LIN {X 0,Y 445.396,Z 554.606,A -85,B 0,C 180,E1 -8729.095,E2 -8729.095} C_VEL
LIN {X 0,Y 445.404,Z 554.809,A -85,B 0,C 180,E1 -8729.999,E2 -8729.999} C_VEL
LIN {X 0,Y 445.396,Z 554.569,A -85,B 0,C 180,E1 -8730.903,E2 -8730.903} C_VEL
LIN {X 0,Y 445.399,Z 553.92,A -85,B 0,C 180,E1 -8731.808,E2 -8731.808} C_VEL
LIN {X 0,Y 445.449,Z 552.858,A -85,B 0,C 180,E1 -8732.712,E2 -8732.712} C_VEL
LIN {X 0,Y 445.409,Z 551.31,A -85,B 0,C 180,E1 -8733.618,E2 -8733.618} C_VEL
LIN {X 0,Y 445.481,Z 548.159,A -85,B 0,C 180,E1 -8734.977,E2 -8734.977} C_VEL
LIN {X 0,Y 445.529,Z 543.719,A -85,B 0,C 180,E1 -8736.385,E2 -8736.385} C_VEL
LIN {X 0,Y 445.7,Z 537.341,A -85,B 0,C 180,E1 -8737.93,E2 -8737.93} C_VEL
LIN {X 0,Y 445.942,Z 530.169,A -85,B 0,C 180,E1 -8739.295,E2 -8739.295} C_VEL
LIN {X 0,Y 446.309,Z 521.18,A -85,B 0,C 180,E1 -8740.662,E2 -8740.662} C_VEL
LIN {X 0,Y 446.885,Z 510.146,A -85,B 0,C 180,E1 -8742.026,E2 -8742.026} C_VEL
LIN {X 0,Y 447.422,Z 499.999,A -85,B 0,C 180,E1 -8743.042,E2 -8743.042} C_VEL
LIN {X 0,Y 447.933,Z 488.57,A -85,B 0,C 180,E1 -8743.958,E2 -8743.958} C_VEL
LIN {X 0,Y 448.567,Z 476.728,A -85,B 0,C 180,E1 -8744.691,E2 -8744.691} C_VEL
LIN {X 0,Y 448.997,Z 463.55,A -85,B 0,C 180,E1 -8745.286,E2 -8745.286} C_VEL
LIN {X 0,Y 449.466,Z 450.413,A -85,B 0,C 180,E1 -8745.676,E2 -8745.676} C_VEL
LIN {X 0,Y 450.087,Z 387.141,A -85,B 0,C 180,E1 -8746.743,E2 -8746.743} C_VEL
LIN {X 0,Y 450.275,Z 363.231,A -85,B 0,C 180,E1 -8747.197,E2 -8747.197} C_VEL
LIN {X 0,Y 447.374,Z 342.684,A -85,B 0,C 180,E1 -8747.702,E2 -8747.702} C_VEL
LIN {X 0,Y 448.31,Z 323.245,A -85,B 0,C 180,E1 -8751.134,E2 -8751.134} C_VEL
LIN {X 0,Y 449.367,Z 304.806,A -85,B 0,C 180,E1 -8754.441,E2 -8754.441} C_VEL
LIN {X 0,Y 447.45,Z 294.39,A -85,B 0,C 180,E1 -8756.454,E2 -8756.454} C_VEL
LIN {X 0,Y 446.525,Z 289.866,A -85,B 0,C 180,E1 -8757.378,E2 -8757.378} C_VEL
LIN {X 0,Y 446.425,Z 289.878,A -85,B 0,C 180,E1 -8760.249,E2 -8760.249} C_VEL
LIN {X 0,Y 446.442,Z 289.872,A -85,B 0,C 180,E1 -8763.453,E2 -8763.453} C_VEL
LIN {X 0,Y 446.396,Z 289.877,A -85,B 0,C 180,E1 -8766.744,E2 -8766.744} C_VEL
LIN {X 0,Y 446.431,Z 289.875,A -85,B 0,C 180,E1 -8770.198,E2 -8770.198} C_VEL
LIN {X 0,Y 446.393,Z 289.881,A -85,B 0,C 180,E1 -8773.596,E2 -8773.596} C_VEL
LIN {X 0,Y 446.391,Z 289.878,A -85,B 0,C 180,E1 -8776.403,E2 -8776.403} C_VEL
LIN {X 0,Y 446.398,Z 289.878,A -85,B 0,C 180,E1 -8779.085,E2 -8779.085} C_VEL
LIN {X 0,Y 446.399,Z 289.878,A -85,B 0,C 180,E1 -8782.12,E2 -8782.12} C_VEL
LIN {X 0,Y 446.416,Z 289.88,A -85,B 0,C 180,E1 -8785.476,E2 -8785.476} C_VEL
LIN {X 0,Y 446.406,Z 289.876,A -85,B 0,C 180,E1 -8788.699,E2 -8788.699} C_VEL
LIN {X 0,Y 446.415,Z 289.877,A -85,B 0,C 180,E1 -8791.836,E2 -8791.836} C_VEL
LIN {X 0,Y 446.422,Z 289.876,A -85,B 0,C 180,E1 -8794.845,E2 -8794.845} C_VEL
LIN {X 0,Y 446.439,Z 289.873,A -85,B 0,C 180,E1 -8798.245,E2 -8798.245} C_VEL
LIN {X 0,Y 446.441,Z 289.874,A -85,B 0,C 180,E1 -8801.648,E2 -8801.648} C_VEL
LIN {X 0,Y 446.495,Z 289.866,A -85,B 0,C 180,E1 -8804.479,E2 -8804.479} C_VEL
LIN {X 0,Y 446.506,Z 289.865,A -85,B 0,C 180,E1 -8808.193,E2 -8808.193} C_VEL
LIN {X 0,Y 446.519,Z 289.867,A -85,B 0,C 180,E1 -8810.944,E2 -8810.944} C_VEL
LIN {X 0,Y 446.588,Z 289.855,A -85,B 0,C 180,E1 -8813.675,E2 -8813.675} C_VEL
LIN {X 0,Y 446.651,Z 289.848,A -85,B 0,C 180,E1 -8817.294,E2 -8817.294} C_VEL
LIN {X 0,Y 446.686,Z 289.843,A -85,B 0,C 180,E1 -8820,E2 -8820} C_VEL
LIN {X 0,Y 446.64,Z 289.851,A -85,B 0,C 180,E1 -8822.706,E2 -8822.706} C_VEL
LIN {X 0,Y 446.595,Z 289.855,A -85,B 0,C 180,E1 -8826.324,E2 -8826.324} C_VEL
LIN {X 0,Y 446.515,Z 289.865,A -85,B 0,C 180,E1 -8829.056,E2 -8829.056} C_VEL
LIN {X 0,Y 446.513,Z 289.867,A -85,B 0,C 180,E1 -8832.73,E2 -8832.73} C_VEL
LIN {X 0,Y 446.479,Z 289.871,A -85,B 0,C 180,E1 -8836.46,E2 -8836.46} C_VEL
LIN {X 0,Y 446.459,Z 289.873,A -85,B 0,C 180,E1 -8839.304,E2 -8839.304} C_VEL
LIN {X 0,Y 446.41,Z 289.879,A -85,B 0,C 180,E1 -8842.2,E2 -8842.2} C_VEL
LIN {X 0,Y 446.431,Z 289.877,A -85,B 0,C 180,E1 -8845.154,E2 -8845.154} C_VEL
LIN {X 0,Y 446.432,Z 289.877,A -85,B 0,C 180,E1 -8848.182,E2 -8848.182} C_VEL
LIN {X 0,Y 446.408,Z 289.879,A -85,B 0,C 180,E1 -8851.301,E2 -8851.301} C_VEL
LIN {X 0,Y 446.422,Z 289.877,A -85,B 0,C 180,E1 -8854.524,E2 -8854.524} C_VEL
LIN {X 0,Y 446.405,Z 289.88,A -85,B 0,C 180,E1 -8858.079,E2 -8858.079} C_VEL
LIN {X 0,Y 446.416,Z 289.879,A -85,B 0,C 180,E1 -8860.918,E2 -8860.918} C_VEL
LIN {X 0,Y 446.393,Z 289.881,A -85,B 0,C 180,E1 -8863.847,E2 -8863.847} C_VEL
LIN {X 0,Y 446.392,Z 289.881,A -85,B 0,C 180,E1 -8866.405,E2 -8866.405} C_VEL
LIN {X 0,Y 446.423,Z 289.876,A -85,B 0,C 180,E1 -8869.083,E2 -8869.083} C_VEL
LIN {X 0,Y 446.405,Z 289.879,A -85,B 0,C 180,E1 -8872.122,E2 -8872.122} C_VEL
LIN {X 0,Y 446.42,Z 289.876,A -85,B 0,C 180,E1 -8875.478,E2 -8875.478} C_VEL
LIN {X 0,Y 446.413,Z 289.879,A -85,B 0,C 180,E1 -8878.701,E2 -8878.701} C_VEL
LIN {X 0,Y 446.483,Z 289.869,A -85,B 0,C 180,E1 -8881.822,E2 -8881.822} C_VEL
LIN {X 0,Y 446.448,Z 289.873,A -85,B 0,C 180,E1 -8884.848,E2 -8884.848} C_VEL
LIN {X 0,Y 446.448,Z 289.875,A -85,B 0,C 180,E1 -8888.246,E2 -8888.246} C_VEL
LIN {X 0,Y 446.519,Z 289.866,A -85,B 0,C 180,E1 -8891.653,E2 -8891.653} C_VEL
LIN {X 0,Y 447.511,Z 295.536,A -85,B 0,C 180,E1 -8892.133,E2 -8892.133} C_VEL
LIN {X 0,Y 451.074,Z 318.693,A -85,B 0,C 180,E1 -8892.665,E2 -8892.665} C_VEL
LIN {X 0,Y 450.362,Z 395.766,A -85,B 0,C 180,E1 -8893.901,E2 -8893.901} C_VEL
LIN {X 0,Y 449.639,Z 401.622,A -85,B 0,C 180,E1 -8893.969,E2 -8893.969} C_VEL
LIN {X 0,Y 445.281,Z 414.821,A -85,B 0,C 180,E1 -8894.091,E2 -8894.091} C_VEL
LIN {X 0,Y 443.656,Z 420.458,A -85,B 0,C 180,E1 -8894.209,E2 -8894.209} C_VEL
LIN {X 0,Y 442.987,Z 426.107,A -85,B 0,C 180,E1 -8894.404,E2 -8894.404} C_VEL
LIN {X 0,Y 442.505,Z 438.201,A -85,B 0,C 180,E1 -8894.986,E2 -8894.986} C_VEL
LIN {X 0,Y 442.002,Z 449.785,A -85,B 0,C 180,E1 -8895.734,E2 -8895.734} C_VEL
LIN {X 0,Y 441.476,Z 461.067,A -85,B 0,C 180,E1 -8896.674,E2 -8896.674} C_VEL
LIN {X 0,Y 440.791,Z 471.918,A -85,B 0,C 180,E1 -8897.805,E2 -8897.805} C_VEL
LIN {X 0,Y 440.215,Z 480.764,A -85,B 0,C 180,E1 -8898.956,E2 -8898.956} C_VEL
LIN {X 0,Y 439.7,Z 489.38,A -85,B 0,C 180,E1 -8900.339,E2 -8900.339} C_VEL
LIN {X 0,Y 439.185,Z 496.313,A -85,B 0,C 180,E1 -8901.72,E2 -8901.72} C_VEL
LIN {X 0,Y 438.904,Z 501.856,A -85,B 0,C 180,E1 -8903.114,E2 -8903.114} C_VEL
LIN {X 0,Y 438.627,Z 506.14,A -85,B 0,C 180,E1 -8904.484,E2 -8904.484} C_VEL
LIN {X 0,Y 438.529,Z 508.41,A -85,B 0,C 180,E1 -8905.405,E2 -8905.405} C_VEL
LIN {X 0,Y 438.578,Z 510.257,A -85,B 0,C 180,E1 -8906.326,E2 -8906.326} C_VEL
LIN {X 0,Y 438.457,Z 511.678,A -85,B 0,C 180,E1 -8907.245,E2 -8907.245} C_VEL
LIN {X 0,Y 438.312,Z 513.288,A -85,B 0,C 180,E1 -8909.082,E2 -8909.082} C_VEL
LIN {X 0,Y 438.314,Z 513.523,A -85,B 0,C 180,E1 -8910.001,E2 -8910.001} C_VEL
LIN {X 0,Y 438.354,Z 512.752,A -85,B 0,C 180,E1 -8911.838,E2 -8911.838} C_VEL
LIN {X 0,Y 438.457,Z 511.788,A -85,B 0,C 180,E1 -8912.757,E2 -8912.757} C_VEL
LIN {X 0,Y 438.572,Z 510.429,A -85,B 0,C 180,E1 -8913.676,E2 -8913.676} C_VEL
LIN {X 0,Y 438.531,Z 507.58,A -85,B 0,C 180,E1 -8915.058,E2 -8915.058} C_VEL
LIN {X 0,Y 438.877,Z 503.69,A -85,B 0,C 180,E1 -8916.437,E2 -8916.437} C_VEL
LIN {X 0,Y 439.039,Z 498.669,A -85,B 0,C 180,E1 -8917.821,E2 -8917.821} C_VEL
LIN {X 0,Y 439.469,Z 492.327,A -85,B 0,C 180,E1 -8919.203,E2 -8919.203} C_VEL
LIN {X 0,Y 439.967,Z 484.438,A -85,B 0,C 180,E1 -8920.586,E2 -8920.586} C_VEL
LIN {X 0,Y 440.452,Z 476.372,A -85,B 0,C 180,E1 -8921.739,E2 -8921.739} C_VEL
LIN {X 0,Y 441.183,Z 466.467,A -85,B 0,C 180,E1 -8922.887,E2 -8922.887} C_VEL
LIN {X 0,Y 441.757,Z 454.932,A -85,B 0,C 180,E1 -8923.96,E2 -8923.96} C_VEL
LIN {X 0,Y 442.266,Z 444.447,A -85,B 0,C 180,E1 -8924.73,E2 -8924.73} C_VEL
LIN {X 0,Y 442.742,Z 432.204,A -85,B 0,C 180,E1 -8925.42,E2 -8925.42} C_VEL
LIN {X 0,Y 443.237,Z 418.659,A -85,B 0,C 180,E1 -8925.963,E2 -8925.963} C_VEL
LIN {X 0,Y 443.407,Z 406.073,A -85,B 0,C 180,E1 -8926.282,E2 -8926.282} C_VEL
LIN {X 0,Y 444.227,Z 319.296,A -85,B 0,C 180,E1 -8927.699,E2 -8927.699} C_VEL
LIN {X 0,Y 440.588,Z 295.599,A -85,B 0,C 180,E1 -8928.263,E2 -8928.263} C_VEL
LIN {X 0,Y 439.49,Z 290.742,A -85,B 0,C 180,E1 -8928.699,E2 -8928.699} C_VEL
LIN {X 0,Y 439.394,Z 290.754,A -85,B 0,C 180,E1 -8931.921,E2 -8931.921} C_VEL
LIN {X 0,Y 439.415,Z 290.749,A -85,B 0,C 180,E1 -8934.573,E2 -8934.573} C_VEL
LIN {X 0,Y 439.445,Z 290.749,A -85,B 0,C 180,E1 -8937.633,E2 -8937.633} C_VEL
LIN {X 0,Y 439.366,Z 290.754,A -85,B 0,C 180,E1 -8940.789,E2 -8940.789} C_VEL
LIN {X 0,Y 439.389,Z 290.752,A -85,B 0,C 180,E1 -8944.044,E2 -8944.044} C_VEL
LIN {X 0,Y 439.353,Z 290.756,A -85,B 0,C 180,E1 -8946.887,E2 -8946.887} C_VEL
LIN {X 0,Y 439.411,Z 290.749,A -85,B 0,C 180,E1 -8949.85,E2 -8949.85} C_VEL
LIN {X 0,Y 439.39,Z 290.751,A -85,B 0,C 180,E1 -8952.628,E2 -8952.628} C_VEL
LIN {X 0,Y 439.407,Z 290.753,A -85,B 0,C 180,E1 -8955.271,E2 -8955.271} C_VEL
LIN {X 0,Y 439.394,Z 290.751,A -85,B 0,C 180,E1 -8958.744,E2 -8958.744} C_VEL
LIN {X 0,Y 439.379,Z 290.752,A -85,B 0,C 180,E1 -8961.608,E2 -8961.608} C_VEL
LIN {X 0,Y 439.404,Z 290.753,A -85,B 0,C 180,E1 -8964.844,E2 -8964.844} C_VEL
LIN {X 0,Y 439.378,Z 290.751,A -85,B 0,C 180,E1 -8968.14,E2 -8968.14} C_VEL
LIN {X 0,Y 439.437,Z 290.744,A -85,B 0,C 180,E1 -8971.598,E2 -8971.598} C_VEL
LIN {X 0,Y 439.393,Z 290.752,A -85,B 0,C 180,E1 -8974.414,E2 -8974.414} C_VEL
LIN {X 0,Y 439.369,Z 290.752,A -85,B 0,C 180,E1 -8977.425,E2 -8977.425} C_VEL
LIN {X 0,Y 439.458,Z 290.872,A -85,B 0,C 180,E1 -8979.247,E2 -8979.247} C_VEL
LIN {X 0,Y 440.572,Z 297.687,A -85,B 0,C 180,E1 -8980.912,E2 -8980.912} C_VEL
LIN {X 0,Y 440.519,Z 303.107,A -85,B 0,C 180,E1 -8982.174,E2 -8982.174} C_VEL
LIN {X 0,Y 443.779,Z 320.199,A -85,B 0,C 180,E1 -8982.629,E2 -8982.629} C_VEL
LIN {X 0,Y 442.424,Z 410.602,A -85,B 0,C 180,E1 -8984.362,E2 -8984.362} C_VEL
LIN {X 0,Y 442.117,Z 424.604,A -85,B 0,C 180,E1 -8984.824,E2 -8984.824} C_VEL
LIN {X 0,Y 441.633,Z 437.177,A -85,B 0,C 180,E1 -8985.426,E2 -8985.426} C_VEL
LIN {X 0,Y 441.219,Z 448.876,A -85,B 0,C 180,E1 -8986.177,E2 -8986.177} C_VEL
LIN {X 0,Y 440.784,Z 460.248,A -85,B 0,C 180,E1 -8987.102,E2 -8987.102} C_VEL
LIN {X 0,Y 440.285,Z 470.498,A -85,B 0,C 180,E1 -8988.14,E2 -8988.14} C_VEL
LIN {X 0,Y 439.756,Z 480.584,A -85,B 0,C 180,E1 -8989.409,E2 -8989.409} C_VEL
LIN {X 0,Y 439.38,Z 488.085,A -85,B 0,C 180,E1 -8990.564,E2 -8990.564} C_VEL
LIN {X 0,Y 438.995,Z 495.45,A -85,B 0,C 180,E1 -8991.947,E2 -8991.947} C_VEL
LIN {X 0,Y 438.781,Z 501.004,A -85,B 0,C 180,E1 -8993.251,E2 -8993.251} C_VEL
LIN {X 0,Y 438.617,Z 505.222,A -85,B 0,C 180,E1 -8994.483,E2 -8994.483} C_VEL
LIN {X 0,Y 438.545,Z 508.87,A -85,B 0,C 180,E1 -8995.864,E2 -8995.864} C_VEL
LIN {X 0,Y 438.457,Z 511.47,A -85,B 0,C 180,E1 -8997.244,E2 -8997.244} C_VEL
LIN {X 0,Y 438.354,Z 512.65,A -85,B 0,C 180,E1 -8998.162,E2 -8998.162} C_VEL
LIN {X 0,Y 438.313,Z 513.401,A -85,B 0,C 180,E1 -8999.081,E2 -8999.081} C_VEL
LIN {X 0,Y 438.317,Z 513.75,A -85,B 0,C 180,E1 -9000,E2 -9000} C_VEL
LIN {X 0,Y 438.342,Z 513.684,A -85,B 0,C 180,E1 -9000.919,E2 -9000.919} C_VEL
LIN {X 0,Y 438.391,Z 513.16,A -85,B 0,C 180,E1 -9001.837,E2 -9001.837} C_VEL
LIN {X 0,Y 438.468,Z 512.228,A -85,B 0,C 180,E1 -9002.756,E2 -9002.756} C_VEL
LIN {X 0,Y 438.588,Z 510.886,A -85,B 0,C 180,E1 -9003.675,E2 -9003.675} C_VEL
LIN {X 0,Y 438.566,Z 508.017,A -85,B 0,C 180,E1 -9005.056,E2 -9005.056} C_VEL
LIN {X 0,Y 438.911,Z 504.057,A -85,B 0,C 180,E1 -9006.436,E2 -9006.436} C_VEL
LIN {X 0,Y 439.14,Z 497.926,A -85,B 0,C 180,E1 -9008.05,E2 -9008.05} C_VEL
LIN {X 0,Y 439.579,Z 491.187,A -85,B 0,C 180,E1 -9009.432,E2 -9009.432} C_VEL
LIN {X 0,Y 440.085,Z 482.787,A -85,B 0,C 180,E1 -9010.815,E2 -9010.815} C_VEL
LIN {X 0,Y 440.469,Z 474.111,A -85,B 0,C 180,E1 -9011.971,E2 -9011.971} C_VEL
LIN {X 0,Y 441.135,Z 463.913,A -85,B 0,C 180,E1 -9013.074,E2 -9013.074} C_VEL
LIN {X 0,Y 441.704,Z 453.145,A -85,B 0,C 180,E1 -9014.019,E2 -9014.019} C_VEL
LIN {X 0,Y 442.222,Z 441.072,A -85,B 0,C 180,E1 -9014.849,E2 -9014.849} C_VEL
LIN {X 0,Y 442.776,Z 427.768,A -85,B 0,C 180,E1 -9015.536,E2 -9015.536} C_VEL
LIN {X 0,Y 443.111,Z 415.088,A -85,B 0,C 180,E1 -9015.996,E2 -9015.996} C_VEL
LIN {X 0,Y 443.534,Z 392.837,A -85,B 0,C 180,E1 -9016.483,E2 -9016.483} C_VEL
LIN {X 0,Y 445.167,Z 320.736,A -85,B 0,C 180,E1 -9017.995,E2 -9017.995} C_VEL
LIN {X 0,Y 441.629,Z 306.236,A -85,B 0,C 180,E1 -9018.559,E2 -9018.559} C_VEL
LIN {X 0,Y 441.447,Z 300.594,A -85,B 0,C 180,E1 -9020.064,E2 -9020.064} C_VEL
LIN {X 0,Y 439.704,Z 292.144,A -85,B 0,C 180,E1 -9022.557,E2 -9022.557} C_VEL
LIN {X 0,Y 439.393,Z 290.755,A -85,B 0,C 180,E1 -9023.009,E2 -9023.009} C_VEL
LIN {X 0,Y 439.37,Z 290.758,A -85,B 0,C 180,E1 -9026.393,E2 -9026.393} C_VEL
LIN {X 0,Y 439.38,Z 290.756,A -85,B 0,C 180,E1 -9028.676,E2 -9028.676} C_VEL
LIN {X 0,Y 439.345,Z 290.758,A -85,B 0,C 180,E1 -9032.024,E2 -9032.024} C_VEL
LIN {X 0,Y 439.385,Z 290.754,A -85,B 0,C 180,E1 -9035.337,E2 -9035.337} C_VEL
LIN {X 0,Y 439.356,Z 290.758,A -85,B 0,C 180,E1 -9038.598,E2 -9038.598} C_VEL
LIN {X 0,Y 439.366,Z 290.755,A -85,B 0,C 180,E1 -9041.252,E2 -9041.252} C_VEL
LIN {X 0,Y 439.377,Z 290.757,A -85,B 0,C 180,E1 -9044.733,E2 -9044.733} C_VEL
LIN {X 0,Y 439.35,Z 290.757,A -85,B 0,C 180,E1 -9047.789,E2 -9047.789} C_VEL
LIN {X 0,Y 439.361,Z 290.755,A -85,B 0,C 180,E1 -9051.402,E2 -9051.402} C_VEL
LIN {X 0,Y 439.401,Z 290.753,A -85,B 0,C 180,E1 -9054.843,E2 -9054.843} C_VEL
LIN {X 0,Y 439.376,Z 290.761,A -85,B 0,C 180,E1 -9058.139,E2 -9058.139} C_VEL
LIN {X 0,Y 439.437,Z 290.78,A -85,B 0,C 180,E1 -9061.327,E2 -9061.327} C_VEL
LIN {X 0,Y 441.863,Z 301.055,A -85,B 0,C 180,E1 -9063.808,E2 -9063.808} C_VEL
LIN {X 0,Y 442.928,Z 307.495,A -85,B 0,C 180,E1 -9065.234,E2 -9065.234} C_VEL
LIN {X 0,Y 441.744,Z 323.154,A -85,B 0,C 180,E1 -9068.29,E2 -9068.29} C_VEL
LIN {X 0,Y 440.732,Z 339.974,A -85,B 0,C 180,E1 -9071.42,E2 -9071.42} C_VEL
LIN {X 0,Y 443.63,Z 357.852,A -85,B 0,C 180,E1 -9071.993,E2 -9071.993} C_VEL
LIN {X 0,Y 444.532,Z 366.532,A -85,B 0,C 180,E1 -9072.239,E2 -9072.239} C_VEL
LIN {X 0,Y 442.866,Z 451.22,A -85,B 0,C 180,E1 -9073.994,E2 -9073.994} C_VEL
LIN {X 0,Y 442.319,Z 464.599,A -85,B 0,C 180,E1 -9074.446,E2 -9074.446} C_VEL
LIN {X 0,Y 441.749,Z 476.41,A -85,B 0,C 180,E1 -9075.016,E2 -9075.016} C_VEL
LIN {X 0,Y 441.114,Z 488.934,A -85,B 0,C 180,E1 -9075.82,E2 -9075.82} C_VEL
LIN {X 0,Y 440.507,Z 499.92,A -85,B 0,C 180,E1 -9076.709,E2 -9076.709} C_VEL
LIN {X 0,Y 439.924,Z 510.52,A -85,B 0,C 180,E1 -9077.779,E2 -9077.779} C_VEL
LIN {X 0,Y 439.448,Z 519.842,A -85,B 0,C 180,E1 -9078.935,E2 -9078.935} C_VEL
LIN {X 0,Y 438.971,Z 528.974,A -85,B 0,C 180,E1 -9080.321,E2 -9080.321} C_VEL
LIN {X 0,Y 438.667,Z 536.272,A -85,B 0,C 180,E1 -9081.709,E2 -9081.709} C_VEL
LIN {X 0,Y 438.46,Z 542.113,A -85,B 0,C 180,E1 -9083.095,E2 -9083.095} C_VEL
LIN {X 0,Y 438.392,Z 546.704,A -85,B 0,C 180,E1 -9084.479,E2 -9084.479} C_VEL
LIN {X 0,Y 438.35,Z 549.141,A -85,B 0,C 180,E1 -9085.401,E2 -9085.401} C_VEL
LIN {X 0,Y 438.294,Z 551.105,A -85,B 0,C 180,E1 -9086.322,E2 -9086.322} C_VEL
LIN {X 0,Y 438.373,Z 552.583,A -85,B 0,C 180,E1 -9087.242,E2 -9087.242} C_VEL
LIN {X 0,Y 438.319,Z 553.638,A -85,B 0,C 180,E1 -9088.161,E2 -9088.161} C_VEL
LIN {X 0,Y 438.306,Z 554.281,A -85,B 0,C 180,E1 -9089.08,E2 -9089.08} C_VEL
LIN {X 0,Y 438.325,Z 554.464,A -85,B 0,C 180,E1 -9089.999,E2 -9089.999} C_VEL
LIN {X 0,Y 438.306,Z 554.212,A -85,B 0,C 180,E1 -9090.918,E2 -9090.918} C_VEL
LIN {X 0,Y 438.319,Z 553.55,A -85,B 0,C 180,E1 -9091.837,E2 -9091.837} C_VEL
LIN {X 0,Y 438.375,Z 552.466,A -85,B 0,C 180,E1 -9092.756,E2 -9092.756} C_VEL
LIN {X 0,Y 438.312,Z 549.968,A -85,B 0,C 180,E1 -9094.137,E2 -9094.137} C_VEL
LIN {X 0,Y 438.383,Z 546.416,A -85,B 0,C 180,E1 -9095.519,E2 -9095.519} C_VEL
LIN {X 0,Y 438.494,Z 541.701,A -85,B 0,C 180,E1 -9096.903,E2 -9096.903} C_VEL
LIN {X 0,Y 438.668,Z 535.673,A -85,B 0,C 180,E1 -9098.289,E2 -9098.289} C_VEL
LIN {X 0,Y 438.94,Z 528.137,A -85,B 0,C 180,E1 -9099.677,E2 -9099.677} C_VEL
LIN {X 0,Y 439.474,Z 517.318,A -85,B 0,C 180,E1 -9101.296,E2 -9101.296} C_VEL
LIN {X 0,Y 439.999,Z 507.714,A -85,B 0,C 180,E1 -9102.452,E2 -9102.452} C_VEL
LIN {X 0,Y 440.662,Z 496.446,A -85,B 0,C 180,E1 -9103.541,E2 -9103.541} C_VEL
LIN {X 0,Y 441.217,Z 484.939,A -85,B 0,C 180,E1 -9104.411,E2 -9104.411} C_VEL
LIN {X 0,Y 441.88,Z 471.957,A -85,B 0,C 180,E1 -9105.154,E2 -9105.154} C_VEL
LIN {X 0,Y 442.338,Z 460.172,A -85,B 0,C 180,E1 -9105.64,E2 -9105.64} C_VEL
LIN {X 0,Y 442.695,Z 447.345,A -85,B 0,C 180,E1 -9105.981,E2 -9105.981} C_VEL
LIN {X 0,Y 443.419,Z 376.801,A -85,B 0,C 180,E1 -9107.158,E2 -9107.158} C_VEL
LIN {X 0,Y 443.415,Z 363.933,A -85,B 0,C 180,E1 -9107.412,E2 -9107.412} C_VEL
LIN {X 0,Y 440.389,Z 342.46,A -85,B 0,C 180,E1 -9107.947,E2 -9107.947} C_VEL
LIN {X 0,Y 441.313,Z 324.12,A -85,B 0,C 180,E1 -9111.24,E2 -9111.24} C_VEL
LIN {X 0,Y 442.378,Z 306.746,A -85,B 0,C 180,E1 -9114.396,E2 -9114.396} C_VEL
LIN {X 0,Y 441.381,Z 299.941,A -85,B 0,C 180,E1 -9115.714,E2 -9115.714} C_VEL
LIN {X 0,Y 439.484,Z 290.743,A -85,B 0,C 180,E1 -9117.564,E2 -9117.564} C_VEL
LIN {X 0,Y 439.358,Z 290.753,A -85,B 0,C 180,E1 -9120.787,E2 -9120.787} C_VEL
LIN {X 0,Y 439.384,Z 290.756,A -85,B 0,C 180,E1 -9124.043,E2 -9124.043} C_VEL
LIN {X 0,Y 439.342,Z 290.755,A -85,B 0,C 180,E1 -9126.886,E2 -9126.886} C_VEL
LIN {X 0,Y 439.397,Z 290.755,A -85,B 0,C 180,E1 -9129.848,E2 -9129.848} C_VEL
LIN {X 0,Y 439.365,Z 290.753,A -85,B 0,C 180,E1 -9132.624,E2 -9132.624} C_VEL
LIN {X 0,Y 439.393,Z 290.751,A -85,B 0,C 180,E1 -9135.269,E2 -9135.269} C_VEL
LIN {X 0,Y 439.364,Z 290.753,A -85,B 0,C 180,E1 -9138.745,E2 -9138.745} C_VEL
LIN {X 0,Y 439.358,Z 290.76,A -85,B 0,C 180,E1 -9141.609,E2 -9141.609} C_VEL
LIN {X 0,Y 439.389,Z 290.75,A -85,B 0,C 180,E1 -9144.843,E2 -9144.843} C_VEL
LIN {X 0,Y 439.364,Z 290.755,A -85,B 0,C 180,E1 -9148.139,E2 -9148.139} C_VEL
LIN {X 0,Y 439.391,Z 290.754,A -85,B 0,C 180,E1 -9151.606,E2 -9151.606} C_VEL
LIN {X 0,Y 439.362,Z 290.754,A -85,B 0,C 180,E1 -9154.412,E2 -9154.412} C_VEL
LIN {X 0,Y 439.353,Z 290.759,A -85,B 0,C 180,E1 -9157.424,E2 -9157.424} C_VEL
LIN {X 0,Y 439.432,Z 290.746,A -85,B 0,C 180,E1 -9160.663,E2 -9160.663} C_VEL
LIN {X 0,Y 439.451,Z 290.744,A -85,B 0,C 180,E1 -9164.224,E2 -9164.224} C_VEL
LIN {X 0,Y 439.473,Z 290.742,A -85,B 0,C 180,E1 -9168.001,E2 -9168.001} C_VEL
LIN {X 0,Y 439.493,Z 290.739,A -85,B 0,C 180,E1 -9171.725,E2 -9171.725} C_VEL
LIN {X 0,Y 439.58,Z 290.728,A -85,B 0,C 180,E1 -9174.495,E2 -9174.495} C_VEL
LIN {X 0,Y 439.619,Z 290.723,A -85,B 0,C 180,E1 -9178.168,E2 -9178.168} C_VEL
LIN {X 0,Y 439.575,Z 290.732,A -85,B 0,C 180,E1 -9180.916,E2 -9180.916} C_VEL
LIN {X 0,Y 439.591,Z 290.73,A -85,B 0,C 180,E1 -9182.749,E2 -9182.749} C_VEL
LIN {X 0,Y 439.548,Z 290.733,A -85,B 0,C 180,E1 -9186.426,E2 -9186.426} C_VEL
LIN {X 0,Y 439.48,Z 290.742,A -85,B 0,C 180,E1 -9189.202,E2 -9189.202} C_VEL
LIN {X 0,Y 439.456,Z 290.745,A -85,B 0,C 180,E1 -9192.938,E2 -9192.938} C_VEL
LIN {X 0,Y 439.437,Z 290.747,A -85,B 0,C 180,E1 -9196.348,E2 -9196.348} C_VEL
LIN {X 0,Y 439.393,Z 290.752,A -85,B 0,C 180,E1 -9199.627,E2 -9199.627} C_VEL
LIN {X 0,Y 439.355,Z 290.758,A -85,B 0,C 180,E1 -9202.576,E2 -9202.576} C_VEL
LIN {X 0,Y 439.37,Z 290.754,A -85,B 0,C 180,E1 -9205.587,E2 -9205.587} C_VEL
LIN {X 0,Y 439.389,Z 290.753,A -85,B 0,C 180,E1 -9208.676,E2 -9208.676} C_VEL
LIN {X 0,Y 439.363,Z 290.756,A -85,B 0,C 180,E1 -9212.031,E2 -9212.031} C_VEL
LIN {X 0,Y 439.386,Z 290.753,A -85,B 0,C 180,E1 -9215.341,E2 -9215.341} C_VEL
LIN {X 0,Y 439.362,Z 290.757,A -85,B 0,C 180,E1 -9218.597,E2 -9218.597} C_VEL
LIN {X 0,Y 439.375,Z 290.754,A -85,B 0,C 180,E1 -9221.257,E2 -9221.257} C_VEL
LIN {X 0,Y 439.393,Z 290.754,A -85,B 0,C 180,E1 -9224.731,E2 -9224.731} C_VEL
LIN {X 0,Y 439.391,Z 290.753,A -85,B 0,C 180,E1 -9227.797,E2 -9227.797} C_VEL
LIN {X 0,Y 439.407,Z 290.751,A -85,B 0,C 180,E1 -9230.227,E2 -9230.227} C_VEL
LIN {X 0,Y 439.37,Z 290.755,A -85,B 0,C 180,E1 -9233.714,E2 -9233.714} C_VEL
LIN {X 0,Y 439.368,Z 290.754,A -85,B 0,C 180,E1 -9237.055,E2 -9237.055} C_VEL
LIN {X 0,Y 439.38,Z 290.755,A -85,B 0,C 180,E1 -9240.275,E2 -9240.275} C_VEL
LIN {X 0,Y 439.427,Z 290.747,A -85,B 0,C 180,E1 -9243.397,E2 -9243.397} C_VEL
LIN {X 0,Y 439.385,Z 290.756,A -85,B 0,C 180,E1 -9246.431,E2 -9246.431} C_VEL
LIN {X 0,Y 439.389,Z 290.753,A -85,B 0,C 180,E1 -9249.398,E2 -9249.398} C_VEL
LIN {X 0,Y 439.466,Z 290.745,A -85,B 0,C 180,E1 -9251.42,E2 -9251.42} C_VEL
LIN {X 0,Y 440.672,Z 296.048,A -85,B 0,C 180,E1 -9251.854,E2 -9251.854} C_VEL
LIN {X 0,Y 444.268,Z 319.368,A -85,B 0,C 180,E1 -9252.398,E2 -9252.398} C_VEL
LIN {X 0,Y 443.349,Z 409.998,A -85,B 0,C 180,E1 -9253.895,E2 -9253.895} C_VEL
LIN {X 0,Y 443.073,Z 423.507,A -85,B 0,C 180,E1 -9254.298,E2 -9254.298} C_VEL
LIN {X 0,Y 442.987,Z 426.107,A -85,B 0,C 180,E1 -9254.404,E2 -9254.404} C_VEL
LIN {X 0,Y 442.25,Z 431.718,A -85,B 0,C 180,E1 -9254.629,E2 -9254.629} C_VEL
LIN {X 0,Y 439.177,Z 440.702,A -85,B 0,C 180,E1 -9255.011,E2 -9255.011} C_VEL
LIN {X 0,Y 435.898,Z 449.345,A -85,B 0,C 180,E1 -9255.474,E2 -9255.474} C_VEL
LIN {X 0,Y 434.895,Z 454.419,A -85,B 0,C 180,E1 -9255.84,E2 -9255.84} C_VEL
LIN {X 0,Y 434.317,Z 465.893,A -85,B 0,C 180,E1 -9256.907,E2 -9256.907} C_VEL
LIN {X 0,Y 433.549,Z 476,A -85,B 0,C 180,E1 -9258.073,E2 -9258.073} C_VEL
LIN {X 0,Y 432.962,Z 485.619,A -85,B 0,C 180,E1 -9259.479,E2 -9259.479} C_VEL
LIN {X 0,Y 432.406,Z 493.357,A -85,B 0,C 180,E1 -9260.883,E2 -9260.883} C_VEL
LIN {X 0,Y 432.05,Z 498.592,A -85,B 0,C 180,E1 -9262.053,E2 -9262.053} C_VEL
LIN {X 0,Y 431.832,Z 503.702,A -85,B 0,C 180,E1 -9263.459,E2 -9263.459} C_VEL
LIN {X 0,Y 431.473,Z 507.664,A -85,B 0,C 180,E1 -9264.861,E2 -9264.861} C_VEL
LIN {X 0,Y 431.495,Z 510.575,A -85,B 0,C 180,E1 -9266.265,E2 -9266.265} C_VEL
LIN {X 0,Y 431.39,Z 511.994,A -85,B 0,C 180,E1 -9267.2,E2 -9267.2} C_VEL
LIN {X 0,Y 431.226,Z 513.604,A -85,B 0,C 180,E1 -9269.067,E2 -9269.067} C_VEL
LIN {X 0,Y 431.225,Z 513.839,A -85,B 0,C 180,E1 -9270.001,E2 -9270.001} C_VEL
LIN {X 0,Y 431.276,Z 513.068,A -85,B 0,C 180,E1 -9271.869,E2 -9271.869} C_VEL
LIN {X 0,Y 431.389,Z 512.103,A -85,B 0,C 180,E1 -9272.802,E2 -9272.802} C_VEL
LIN {X 0,Y 431.489,Z 510.744,A -85,B 0,C 180,E1 -9273.736,E2 -9273.736} C_VEL
LIN {X 0,Y 431.471,Z 507.895,A -85,B 0,C 180,E1 -9275.141,E2 -9275.141} C_VEL
LIN {X 0,Y 431.809,Z 504.005,A -85,B 0,C 180,E1 -9276.543,E2 -9276.543} C_VEL
LIN {X 0,Y 432.022,Z 498.981,A -85,B 0,C 180,E1 -9277.949,E2 -9277.949} C_VEL
LIN {X 0,Y 432.474,Z 492.638,A -85,B 0,C 180,E1 -9279.353,E2 -9279.353} C_VEL
LIN {X 0,Y 432.997,Z 484.746,A -85,B 0,C 180,E1 -9280.759,E2 -9280.759} C_VEL
LIN {X 0,Y 433.522,Z 476.678,A -85,B 0,C 180,E1 -9281.93,E2 -9281.93} C_VEL
LIN {X 0,Y 434.286,Z 466.768,A -85,B 0,C 180,E1 -9283.096,E2 -9283.096} C_VEL
LIN {X 0,Y 434.853,Z 455.78,A -85,B 0,C 180,E1 -9284.138,E2 -9284.138} C_VEL
LIN {X 0,Y 435.417,Z 444.736,A -85,B 0,C 180,E1 -9284.967,E2 -9284.967} C_VEL
LIN {X 0,Y 435.924,Z 432.478,A -85,B 0,C 180,E1 -9285.668,E2 -9285.668} C_VEL
LIN {X 0,Y 436.417,Z 419.742,A -85,B 0,C 180,E1 -9286.189,E2 -9286.189} C_VEL
LIN {X 0,Y 436.628,Z 407.793,A -85,B 0,C 180,E1 -9286.512,E2 -9286.512} C_VEL
LIN {X 0,Y 437.477,Z 319.891,A -85,B 0,C 180,E1 -9287.974,E2 -9287.974} C_VEL
LIN {X 0,Y 433.744,Z 296.583,A -85,B 0,C 180,E1 -9288.537,E2 -9288.537} C_VEL
LIN {X 0,Y 432.439,Z 291.679,A -85,B 0,C 180,E1 -9288.919,E2 -9288.919} C_VEL
LIN {X 0,Y 432.349,Z 291.63,A -85,B 0,C 180,E1 -9292.095,E2 -9292.095} C_VEL
LIN {X 0,Y 432.351,Z 291.628,A -85,B 0,C 180,E1 -9295.002,E2 -9295.002} C_VEL
LIN {X 0,Y 432.386,Z 291.625,A -85,B 0,C 180,E1 -9298.124,E2 -9298.124} C_VEL
LIN {X 0,Y 432.325,Z 291.634,A -85,B 0,C 180,E1 -9301.347,E2 -9301.347} C_VEL
LIN {X 0,Y 432.342,Z 291.628,A -85,B 0,C 180,E1 -9304.678,E2 -9304.678} C_VEL
LIN {X 0,Y 432.343,Z 291.629,A -85,B 0,C 180,E1 -9308.15,E2 -9308.15} C_VEL
LIN {X 0,Y 432.338,Z 291.631,A -85,B 0,C 180,E1 -9311.602,E2 -9311.602} C_VEL
LIN {X 0,Y 432.345,Z 291.627,A -85,B 0,C 180,E1 -9314.347,E2 -9314.347} C_VEL
LIN {X 0,Y 432.325,Z 291.634,A -85,B 0,C 180,E1 -9317.016,E2 -9317.016} C_VEL
LIN {X 0,Y 432.338,Z 291.629,A -85,B 0,C 180,E1 -9319.821,E2 -9319.821} C_VEL
LIN {X 0,Y 432.312,Z 291.638,A -85,B 0,C 180,E1 -9323.022,E2 -9323.022} C_VEL
LIN {X 0,Y 432.364,Z 291.625,A -85,B 0,C 180,E1 -9325.997,E2 -9325.997} C_VEL
LIN {X 0,Y 432.352,Z 291.627,A -85,B 0,C 180,E1 -9329.49,E2 -9329.49} C_VEL
LIN {X 0,Y 432.39,Z 291.626,A -85,B 0,C 180,E1 -9332.928,E2 -9332.928} C_VEL
LIN {X 0,Y 432.372,Z 291.624,A -85,B 0,C 180,E1 -9336.023,E2 -9336.023} C_VEL
LIN {X 0,Y 432.417,Z 291.788,A -85,B 0,C 180,E1 -9339.112,E2 -9339.112} C_VEL
LIN {X 0,Y 433.645,Z 299.803,A -85,B 0,C 180,E1 -9341.087,E2 -9341.087} C_VEL
LIN {X 0,Y 433.562,Z 303.369,A -85,B 0,C 180,E1 -9341.924,E2 -9341.924} C_VEL
LIN {X 0,Y 436.906,Z 321.998,A -85,B 0,C 180,E1 -9342.425,E2 -9342.425} C_VEL
LIN {X 0,Y 435.475,Z 411.691,A -85,B 0,C 180,E1 -9344.196,E2 -9344.196} C_VEL
LIN {X 0,Y 435.162,Z 425.405,A -85,B 0,C 180,E1 -9344.665,E2 -9344.665} C_VEL
LIN {X 0,Y 434.669,Z 437.301,A -85,B 0,C 180,E1 -9345.247,E2 -9345.247} C_VEL
LIN {X 0,Y 434.212,Z 450.31,A -85,B 0,C 180,E1 -9346.104,E2 -9346.104} C_VEL
LIN {X 0,Y 433.754,Z 461.089,A -85,B 0,C 180,E1 -9347.008,E2 -9347.008} C_VEL
LIN {X 0,Y 433.252,Z 471.224,A -85,B 0,C 180,E1 -9348.064,E2 -9348.064} C_VEL
LIN {X 0,Y 432.724,Z 480.421,A -85,B 0,C 180,E1 -9349.235,E2 -9349.235} C_VEL
LIN {X 0,Y 432.287,Z 489.401,A -85,B 0,C 180,E1 -9350.643,E2 -9350.643} C_VEL
LIN {X 0,Y 431.905,Z 496.537,A -85,B 0,C 180,E1 -9352.05,E2 -9352.05} C_VEL
LIN {X 0,Y 431.702,Z 502.243,A -85,B 0,C 180,E1 -9353.456,E2 -9353.456} C_VEL
LIN {X 0,Y 431.463,Z 506.706,A -85,B 0,C 180,E1 -9354.86,E2 -9354.86} C_VEL
LIN {X 0,Y 431.454,Z 510.047,A -85,B 0,C 180,E1 -9356.264,E2 -9356.264} C_VEL
LIN {X 0,Y 431.388,Z 511.719,A -85,B 0,C 180,E1 -9357.199,E2 -9357.199} C_VEL
LIN {X 0,Y 431.276,Z 512.942,A -85,B 0,C 180,E1 -9358.132,E2 -9358.132} C_VEL
LIN {X 0,Y 431.227,Z 513.715,A -85,B 0,C 180,E1 -9359.066,E2 -9359.066} C_VEL
LIN {X 0,Y 431.228,Z 514.086,A -85,B 0,C 180,E1 -9360,E2 -9360} C_VEL
LIN {X 0,Y 431.255,Z 514.048,A -85,B 0,C 180,E1 -9360.934,E2 -9360.934} C_VEL
LIN {X 0,Y 431.31,Z 513.549,A -85,B 0,C 180,E1 -9361.868,E2 -9361.868} C_VEL
LIN {X 0,Y 431.4,Z 512.631,A -85,B 0,C 180,E1 -9362.801,E2 -9362.801} C_VEL
LIN {X 0,Y 431.528,Z 511.305,A -85,B 0,C 180,E1 -9363.735,E2 -9363.735} C_VEL
LIN {X 0,Y 431.5,Z 508.469,A -85,B 0,C 180,E1 -9365.139,E2 -9365.139} C_VEL
LIN {X 0,Y 431.873,Z 504.539,A -85,B 0,C 180,E1 -9366.541,E2 -9366.541} C_VEL
LIN {X 0,Y 432.081,Z 499.45,A -85,B 0,C 180,E1 -9367.947,E2 -9367.947} C_VEL
LIN {X 0,Y 432.523,Z 492.98,A -85,B 0,C 180,E1 -9369.351,E2 -9369.351} C_VEL
LIN {X 0,Y 433.049,Z 484.897,A -85,B 0,C 180,E1 -9370.756,E2 -9370.756} C_VEL
LIN {X 0,Y 433.505,Z 476.637,A -85,B 0,C 180,E1 -9371.929,E2 -9371.929} C_VEL
LIN {X 0,Y 434.163,Z 466.5,A -85,B 0,C 180,E1 -9373.098,E2 -9373.098} C_VEL
LIN {X 0,Y 434.811,Z 455.525,A -85,B 0,C 180,E1 -9374.114,E2 -9374.114} C_VEL
LIN {X 0,Y 435.389,Z 443.971,A -85,B 0,C 180,E1 -9374.967,E2 -9374.967} C_VEL
LIN {X 0,Y 435.938,Z 431.516,A -85,B 0,C 180,E1 -9375.666,E2 -9375.666} C_VEL
LIN {X 0,Y 436.362,Z 418.694,A -85,B 0,C 180,E1 -9376.191,E2 -9376.191} C_VEL
LIN {X 0,Y 436.642,Z 405.669,A -85,B 0,C 180,E1 -9376.54,E2 -9376.54} C_VEL
LIN {X 0,Y 438.533,Z 326.572,A -85,B 0,C 180,E1 -9378.238,E2 -9378.238} C_VEL
LIN {X 0,Y 438.515,Z 321.194,A -85,B 0,C 180,E1 -9378.368,E2 -9378.368} C_VEL
LIN {X 0,Y 434.839,Z 306.813,A -85,B 0,C 180,E1 -9378.951,E2 -9378.951} C_VEL
LIN {X 0,Y 434.564,Z 302.02,A -85,B 0,C 180,E1 -9380.279,E2 -9380.279} C_VEL
LIN {X 0,Y 432.718,Z 293.276,A -85,B 0,C 180,E1 -9382.942,E2 -9382.942} C_VEL
LIN {X 0,Y 432.352,Z 291.633,A -85,B 0,C 180,E1 -9383.469,E2 -9383.469} C_VEL
LIN {X 0,Y 432.313,Z 291.637,A -85,B 0,C 180,E1 -9386.603,E2 -9386.603} C_VEL
LIN {X 0,Y 432.318,Z 291.636,A -85,B 0,C 180,E1 -9389.189,E2 -9389.189} C_VEL
LIN {X 0,Y 432.308,Z 291.636,A -85,B 0,C 180,E1 -9392.444,E2 -9392.444} C_VEL
LIN {X 0,Y 432.333,Z 291.631,A -85,B 0,C 180,E1 -9395.818,E2 -9395.818} C_VEL
LIN {X 0,Y 432.303,Z 291.635,A -85,B 0,C 180,E1 -9399.348,E2 -9399.348} C_VEL
LIN {X 0,Y 432.306,Z 291.634,A -85,B 0,C 180,E1 -9401.801,E2 -9401.801} C_VEL
LIN {X 0,Y 432.335,Z 291.632,A -85,B 0,C 180,E1 -9404.347,E2 -9404.347} C_VEL
LIN {X 0,Y 432.304,Z 291.635,A -85,B 0,C 180,E1 -9407.018,E2 -9407.018} C_VEL
LIN {X 0,Y 432.292,Z 291.637,A -85,B 0,C 180,E1 -9409.828,E2 -9409.828} C_VEL
LIN {X 0,Y 432.306,Z 291.636,A -85,B 0,C 180,E1 -9413.021,E2 -9413.021} C_VEL
LIN {X 0,Y 432.363,Z 291.631,A -85,B 0,C 180,E1 -9415.996,E2 -9415.996} C_VEL
LIN {X 0,Y 432.35,Z 291.637,A -85,B 0,C 180,E1 -9419.489,E2 -9419.489} C_VEL
LIN {X 0,Y 432.386,Z 291.75,A -85,B 0,C 180,E1 -9420.854,E2 -9420.854} C_VEL
LIN {X 0,Y 434.5,Z 300.489,A -85,B 0,C 180,E1 -9423.069,E2 -9423.069} C_VEL
LIN {X 0,Y 436.059,Z 308.799,A -85,B 0,C 180,E1 -9424.996,E2 -9424.996} C_VEL
LIN {X 0,Y 435.324,Z 318.485,A -85,B 0,C 180,E1 -9426.959,E2 -9426.959} C_VEL
LIN {X 0,Y 434.2,Z 333.348,A -85,B 0,C 180,E1 -9429.85,E2 -9429.85} C_VEL
LIN {X 0,Y 433.877,Z 339.369,A -85,B 0,C 180,E1 -9430.993,E2 -9430.993} C_VEL
LIN {X 0,Y 436.844,Z 356.926,A -85,B 0,C 180,E1 -9431.599,E2 -9431.599} C_VEL
LIN {X 0,Y 437.939,Z 367.347,A -85,B 0,C 180,E1 -9431.908,E2 -9431.908} C_VEL
LIN {X 0,Y 436.125,Z 450.293,A -85,B 0,C 180,E1 -9433.679,E2 -9433.679} C_VEL
LIN {X 0,Y 435.57,Z 463.723,A -85,B 0,C 180,E1 -9434.139,E2 -9434.139} C_VEL
LIN {X 0,Y 434.902,Z 476.616,A -85,B 0,C 180,E1 -9434.775,E2 -9434.775} C_VEL
LIN {X 0,Y 434.228,Z 489.007,A -85,B 0,C 180,E1 -9435.59,E2 -9435.59} C_VEL
LIN {X 0,Y 433.535,Z 500.715,A -85,B 0,C 180,E1 -9436.571,E2 -9436.571} C_VEL
LIN {X 0,Y 432.909,Z 511.4,A -85,B 0,C 180,E1 -9437.696,E2 -9437.696} C_VEL
LIN {X 0,Y 432.331,Z 521.361,A -85,B 0,C 180,E1 -9438.987,E2 -9438.987} C_VEL
LIN {X 0,Y 431.862,Z 530.071,A -85,B 0,C 180,E1 -9440.397,E2 -9440.397} C_VEL
LIN {X 0,Y 431.579,Z 537.099,A -85,B 0,C 180,E1 -9441.807,E2 -9441.807} C_VEL
LIN {X 0,Y 431.34,Z 543.533,A -85,B 0,C 180,E1 -9443.45,E2 -9443.45} C_VEL
LIN {X 0,Y 431.306,Z 547.722,A -85,B 0,C 180,E1 -9444.857,E2 -9444.857} C_VEL
LIN {X 0,Y 431.2,Z 550.81,A -85,B 0,C 180,E1 -9446.261,E2 -9446.261} C_VEL
LIN {X 0,Y 431.281,Z 552.28,A -85,B 0,C 180,E1 -9447.197,E2 -9447.197} C_VEL
LIN {X 0,Y 431.241,Z 553.326,A -85,B 0,C 180,E1 -9448.131,E2 -9448.131} C_VEL
LIN {X 0,Y 431.22,Z 553.955,A -85,B 0,C 180,E1 -9449.065,E2 -9449.065} C_VEL
LIN {X 0,Y 431.235,Z 554.115,A -85,B 0,C 180,E1 -9449.999,E2 -9449.999} C_VEL
LIN {X 0,Y 431.22,Z 553.851,A -85,B 0,C 180,E1 -9450.933,E2 -9450.933} C_VEL
LIN {X 0,Y 431.241,Z 553.174,A -85,B 0,C 180,E1 -9451.867,E2 -9451.867} C_VEL
LIN {X 0,Y 431.302,Z 552.059,A -85,B 0,C 180,E1 -9452.801,E2 -9452.801} C_VEL
LIN {X 0,Y 431.229,Z 549.523,A -85,B 0,C 180,E1 -9454.205,E2 -9454.205} C_VEL
LIN {X 0,Y 431.286,Z 545.921,A -85,B 0,C 180,E1 -9455.61,E2 -9455.61} C_VEL
LIN {X 0,Y 431.413,Z 541.145,A -85,B 0,C 180,E1 -9457.017,E2 -9457.017} C_VEL
LIN {X 0,Y 431.609,Z 535.053,A -85,B 0,C 180,E1 -9458.426,E2 -9458.426} C_VEL
LIN {X 0,Y 431.995,Z 524.847,A -85,B 0,C 180,E1 -9460.308,E2 -9460.308} C_VEL
LIN {X 0,Y 432.48,Z 517.004,A -85,B 0,C 180,E1 -9461.481,E2 -9461.481} C_VEL
LIN {X 0,Y 433.036,Z 507.402,A -85,B 0,C 180,E1 -9462.655,E2 -9462.655} C_VEL
LIN {X 0,Y 433.702,Z 496.516,A -85,B 0,C 180,E1 -9463.728,E2 -9463.728} C_VEL
LIN {X 0,Y 434.244,Z 486.378,A -85,B 0,C 180,E1 -9464.527,E2 -9464.527} C_VEL
LIN {X 0,Y 434.892,Z 473.905,A -85,B 0,C 180,E1 -9465.284,E2 -9465.284} C_VEL
LIN {X 0,Y 435.431,Z 460.728,A -85,B 0,C 180,E1 -9465.864,E2 -9465.864} C_VEL
LIN {X 0,Y 435.852,Z 448.572,A -85,B 0,C 180,E1 -9466.209,E2 -9466.209} C_VEL
LIN {X 0,Y 436.633,Z 365.258,A -85,B 0,C 180,E1 -9467.612,E2 -9467.612} C_VEL
LIN {X 0,Y 433.411,Z 342.095,A -85,B 0,C 180,E1 -9468.218,E2 -9468.218} C_VEL
LIN {X 0,Y 434.36,Z 323.578,A -85,B 0,C 180,E1 -9471.597,E2 -9471.597} C_VEL
LIN {X 0,Y 435.401,Z 307.567,A -85,B 0,C 180,E1 -9474.559,E2 -9474.559} C_VEL
LIN {X 0,Y 434.038,Z 299.436,A -85,B 0,C 180,E1 -9476.175,E2 -9476.175} C_VEL
LIN {X 0,Y 432.433,Z 291.622,A -85,B 0,C 180,E1 -9477.789,E2 -9477.789} C_VEL
LIN {X 0,Y 432.318,Z 291.63,A -85,B 0,C 180,E1 -9481.345,E2 -9481.345} C_VEL
LIN {X 0,Y 432.335,Z 291.629,A -85,B 0,C 180,E1 -9484.676,E2 -9484.676} C_VEL
LIN {X 0,Y 432.327,Z 291.633,A -85,B 0,C 180,E1 -9488.149,E2 -9488.149} C_VEL
LIN {X 0,Y 432.319,Z 291.634,A -85,B 0,C 180,E1 -9491.6,E2 -9491.6} C_VEL
LIN {X 0,Y 432.328,Z 291.631,A -85,B 0,C 180,E1 -9494.346,E2 -9494.346} C_VEL
LIN {X 0,Y 432.31,Z 291.632,A -85,B 0,C 180,E1 -9497.015,E2 -9497.015} C_VEL
LIN {X 0,Y 432.284,Z 291.64,A -85,B 0,C 180,E1 -9499.827,E2 -9499.827} C_VEL
LIN {X 0,Y 432.299,Z 291.634,A -85,B 0,C 180,E1 -9503.021,E2 -9503.021} C_VEL
LIN {X 0,Y 432.35,Z 291.629,A -85,B 0,C 180,E1 -9505.996,E2 -9505.996} C_VEL
LIN {X 0,Y 432.338,Z 291.634,A -85,B 0,C 180,E1 -9509.489,E2 -9509.489} C_VEL
LIN {X 0,Y 432.319,Z 291.633,A -85,B 0,C 180,E1 -9511.872,E2 -9511.872} C_VEL
LIN {X 0,Y 432.356,Z 291.63,A -85,B 0,C 180,E1 -9515.542,E2 -9515.542} C_VEL
LIN {X 0,Y 432.341,Z 291.631,A -85,B 0,C 180,E1 -9519.046,E2 -9519.046} C_VEL
LIN {X 0,Y 432.35,Z 291.629,A -85,B 0,C 180,E1 -9522.01,E2 -9522.01} C_VEL
LIN {X 0,Y 432.38,Z 291.626,A -85,B 0,C 180,E1 -9524.926,E2 -9524.926} C_VEL
LIN {X 0,Y 432.449,Z 291.617,A -85,B 0,C 180,E1 -9527.803,E2 -9527.803} C_VEL
LIN {X 0,Y 432.453,Z 291.617,A -85,B 0,C 180,E1 -9531.59,E2 -9531.59} C_VEL
LIN {X 0,Y 432.536,Z 291.605,A -85,B 0,C 180,E1 -9534.405,E2 -9534.405} C_VEL
LIN {X 0,Y 432.588,Z 291.598,A -85,B 0,C 180,E1 -9538.138,E2 -9538.138} C_VEL
LIN {X 0,Y 432.536,Z 291.609,A -85,B 0,C 180,E1 -9540.931,E2 -9540.931} C_VEL
LIN {X 0,Y 432.545,Z 291.608,A -85,B 0,C 180,E1 -9542.794,E2 -9542.794} C_VEL
LIN {X 0,Y 432.505,Z 291.611,A -85,B 0,C 180,E1 -9546.531,E2 -9546.531} C_VEL
LIN {X 0,Y 432.424,Z 291.621,A -85,B 0,C 180,E1 -9549.354,E2 -9549.354} C_VEL
LIN {X 0,Y 432.422,Z 291.622,A -85,B 0,C 180,E1 -9552.804,E2 -9552.804} C_VEL
LIN {X 0,Y 432.403,Z 291.624,A -85,B 0,C 180,E1 -9556.479,E2 -9556.479} C_VEL
LIN {X 0,Y 432.329,Z 291.631,A -85,B 0,C 180,E1 -9559.961,E2 -9559.961} C_VEL
LIN {X 0,Y 432.309,Z 291.635,A -85,B 0,C 180,E1 -9562.965,E2 -9562.965} C_VEL
LIN {X 0,Y 432.33,Z 291.633,A -85,B 0,C 180,E1 -9565.003,E2 -9565.003} C_VEL
LIN {X 0,Y 432.336,Z 291.632,A -85,B 0,C 180,E1 -9568.127,E2 -9568.127} C_VEL
LIN {X 0,Y 432.313,Z 291.634,A -85,B 0,C 180,E1 -9571.347,E2 -9571.347} C_VEL
LIN {X 0,Y 432.332,Z 291.632,A -85,B 0,C 180,E1 -9574.678,E2 -9574.678} C_VEL
LIN {X 0,Y 432.325,Z 291.634,A -85,B 0,C 180,E1 -9578.151,E2 -9578.151} C_VEL
LIN {X 0,Y 432.318,Z 291.632,A -85,B 0,C 180,E1 -9581.602,E2 -9581.602} C_VEL
LIN {X 0,Y 432.328,Z 291.633,A -85,B 0,C 180,E1 -9584.348,E2 -9584.348} C_VEL
LIN {X 0,Y 432.315,Z 291.634,A -85,B 0,C 180,E1 -9587.017,E2 -9587.017} C_VEL
LIN {X 0,Y 432.329,Z 291.633,A -85,B 0,C 180,E1 -9589.822,E2 -9589.822} C_VEL
LIN {X 0,Y 432.303,Z 291.635,A -85,B 0,C 180,E1 -9593.023,E2 -9593.023} C_VEL
LIN {X 0,Y 432.354,Z 291.629,A -85,B 0,C 180,E1 -9595.998,E2 -9595.998} C_VEL
LIN {X 0,Y 432.345,Z 291.629,A -85,B 0,C 180,E1 -9599.491,E2 -9599.491} C_VEL
LIN {X 0,Y 432.389,Z 291.624,A -85,B 0,C 180,E1 -9602.929,E2 -9602.929} C_VEL
LIN {X 0,Y 432.369,Z 291.628,A -85,B 0,C 180,E1 -9606.024,E2 -9606.024} C_VEL
LIN {X 0,Y 432.351,Z 291.632,A -85,B 0,C 180,E1 -9609.047,E2 -9609.047} C_VEL
LIN {X 0,Y 432.409,Z 291.625,A -85,B 0,C 180,E1 -9611.166,E2 -9611.166} C_VEL
LIN {X 0,Y 433.755,Z 296.538,A -85,B 0,C 180,E1 -9611.559,E2 -9611.559} C_VEL
LIN {X 0,Y 437.387,Z 319.251,A -85,B 0,C 180,E1 -9612.106,E2 -9612.106} C_VEL
LIN {X 0,Y 436.695,Z 402.694,A -85,B 0,C 180,E1 -9613.493,E2 -9613.493} C_VEL
LIN {X 0,Y 436.45,Z 416.9,A -85,B 0,C 180,E1 -9613.814,E2 -9613.814} C_VEL
LIN {X 0,Y 436.055,Z 429.381,A -85,B 0,C 180,E1 -9614.279,E2 -9614.279} C_VEL
LIN {X 0,Y 435.563,Z 441.427,A -85,B 0,C 180,E1 -9614.92,E2 -9614.92} C_VEL
LIN {X 0,Y 434.965,Z 453.411,A -85,B 0,C 180,E1 -9615.76,E2 -9615.76} C_VEL
LIN {X 0,Y 434.895,Z 454.419,A -85,B 0,C 180,E1 -9615.84,E2 -9615.84} C_VEL
LIN {X 0,Y 433.915,Z 459.418,A -85,B 0,C 180,E1 -9616.238,E2 -9616.238} C_VEL
LIN {X 0,Y 430.624,Z 467.269,A -85,B 0,C 180,E1 -9616.916,E2 -9616.916} C_VEL
LIN {X 0,Y 427.372,Z 474.659,A -85,B 0,C 180,E1 -9617.687,E2 -9617.687} C_VEL
LIN {X 0,Y 426.46,Z 478.857,A -85,B 0,C 180,E1 -9618.226,E2 -9618.226} C_VEL
LIN {X 0,Y 425.904,Z 487.369,A -85,B 0,C 180,E1 -9619.543,E2 -9619.543} C_VEL
LIN {X 0,Y 425.303,Z 494.786,A -85,B 0,C 180,E1 -9620.969,E2 -9620.969} C_VEL
LIN {X 0,Y 424.901,Z 500.739,A -85,B 0,C 180,E1 -9622.397,E2 -9622.397} C_VEL
LIN {X 0,Y 424.71,Z 505.44,A -85,B 0,C 180,E1 -9623.826,E2 -9623.826} C_VEL
LIN {X 0,Y 424.367,Z 509.045,A -85,B 0,C 180,E1 -9625.251,E2 -9625.251} C_VEL
LIN {X 0,Y 424.415,Z 510.892,A -85,B 0,C 180,E1 -9626.203,E2 -9626.203} C_VEL
LIN {X 0,Y 424.324,Z 512.31,A -85,B 0,C 180,E1 -9627.153,E2 -9627.153} C_VEL
LIN {X 0,Y 424.143,Z 513.921,A -85,B 0,C 180,E1 -9629.052,E2 -9629.052} C_VEL
LIN {X 0,Y 424.139,Z 514.156,A -85,B 0,C 180,E1 -9630.001,E2 -9630.001} C_VEL
LIN {X 0,Y 424.201,Z 513.383,A -85,B 0,C 180,E1 -9631.9,E2 -9631.9} C_VEL
LIN {X 0,Y 424.323,Z 512.418,A -85,B 0,C 180,E1 -9632.849,E2 -9632.849} C_VEL
LIN {X 0,Y 424.409,Z 511.06,A -85,B 0,C 180,E1 -9633.799,E2 -9633.799} C_VEL
LIN {X 0,Y 424.417,Z 508.209,A -85,B 0,C 180,E1 -9635.226,E2 -9635.226} C_VEL
LIN {X 0,Y 424.735,Z 504.32,A -85,B 0,C 180,E1 -9636.652,E2 -9636.652} C_VEL
LIN {X 0,Y 424.982,Z 499.294,A -85,B 0,C 180,E1 -9638.082,E2 -9638.082} C_VEL
LIN {X 0,Y 425.482,Z 492.949,A -85,B 0,C 180,E1 -9639.508,E2 -9639.508} C_VEL
LIN {X 0,Y 426.015,Z 485.056,A -85,B 0,C 180,E1 -9640.937,E2 -9640.937} C_VEL
LIN {X 0,Y 426.6,Z 476.983,A -85,B 0,C 180,E1 -9642.126,E2 -9642.126} C_VEL
LIN {X 0,Y 427.386,Z 467.07,A -85,B 0,C 180,E1 -9643.311,E2 -9643.311} C_VEL
LIN {X 0,Y 427.928,Z 456.791,A -85,B 0,C 180,E1 -9644.308,E2 -9644.308} C_VEL
LIN {X 0,Y 428.583,Z 445.025,A -85,B 0,C 180,E1 -9645.212,E2 -9645.212} C_VEL
LIN {X 0,Y 429.115,Z 432.752,A -85,B 0,C 180,E1 -9645.923,E2 -9645.923} C_VEL
LIN {X 0,Y 429.631,Z 419.995,A -85,B 0,C 180,E1 -9646.452,E2 -9646.452} C_VEL
LIN {X 0,Y 429.852,Z 407.996,A -85,B 0,C 180,E1 -9646.78,E2 -9646.78} C_VEL
LIN {X 0,Y 430.693,Z 320.419,A -85,B 0,C 180,E1 -9648.261,E2 -9648.261} C_VEL
LIN {X 0,Y 427.188,Z 298.403,A -85,B 0,C 180,E1 -9648.803,E2 -9648.803} C_VEL
LIN {X 0,Y 426.23,Z 295.552,A -85,B 0,C 180,E1 -9648.93,E2 -9648.93} C_VEL
LIN {X 0,Y 425.368,Z 292.502,A -85,B 0,C 180,E1 -9649.224,E2 -9649.224} C_VEL
LIN {X 0,Y 425.293,Z 292.509,A -85,B 0,C 180,E1 -9652.339,E2 -9652.339} C_VEL
LIN {X 0,Y 425.296,Z 292.509,A -85,B 0,C 180,E1 -9655.446,E2 -9655.446} C_VEL
LIN {X 0,Y 425.353,Z 292.503,A -85,B 0,C 180,E1 -9657.558,E2 -9657.558} C_VEL
LIN {X 0,Y 425.293,Z 292.506,A -85,B 0,C 180,E1 -9660.817,E2 -9660.817} C_VEL
LIN {X 0,Y 425.314,Z 292.504,A -85,B 0,C 180,E1 -9664.288,E2 -9664.288} C_VEL
LIN {X 0,Y 425.284,Z 292.51,A -85,B 0,C 180,E1 -9667.695,E2 -9667.695} C_VEL
LIN {X 0,Y 425.286,Z 292.507,A -85,B 0,C 180,E1 -9670.521,E2 -9670.521} C_VEL
LIN {X 0,Y 425.269,Z 292.514,A -85,B 0,C 180,E1 -9673.352,E2 -9673.352} C_VEL
LIN {X 0,Y 425.263,Z 292.511,A -85,B 0,C 180,E1 -9676.649,E2 -9676.649} C_VEL
LIN {X 0,Y 425.292,Z 292.507,A -85,B 0,C 180,E1 -9679.873,E2 -9679.873} C_VEL
LIN {X 0,Y 425.283,Z 292.508,A -85,B 0,C 180,E1 -9682.489,E2 -9682.489} C_VEL
LIN {X 0,Y 425.312,Z 292.503,A -85,B 0,C 180,E1 -9685.818,E2 -9685.818} C_VEL
LIN {X 0,Y 425.296,Z 292.508,A -85,B 0,C 180,E1 -9689.239,E2 -9689.239} C_VEL
LIN {X 0,Y 425.35,Z 292.501,A -85,B 0,C 180,E1 -9692.442,E2 -9692.442} C_VEL
LIN {X 0,Y 425.352,Z 292.498,A -85,B 0,C 180,E1 -9695.602,E2 -9695.602} C_VEL
LIN {X 0,Y 425.365,Z 292.552,A -85,B 0,C 180,E1 -9698.939,E2 -9698.939} C_VEL
LIN {X 0,Y 426.667,Z 300.889,A -85,B 0,C 180,E1 -9701.015,E2 -9701.015} C_VEL
LIN {X 0,Y 426.599,Z 303.623,A -85,B 0,C 180,E1 -9701.666,E2 -9701.666} C_VEL
LIN {X 0,Y 430.037,Z 322.159,A -85,B 0,C 180,E1 -9702.189,E2 -9702.189} C_VEL
LIN {X 0,Y 428.539,Z 411.49,A -85,B 0,C 180,E1 -9703.995,E2 -9703.995} C_VEL
LIN {X 0,Y 428.23,Z 425.321,A -85,B 0,C 180,E1 -9704.471,E2 -9704.471} C_VEL
LIN {X 0,Y 427.716,Z 437.33,A -85,B 0,C 180,E1 -9705.062,E2 -9705.062} C_VEL
LIN {X 0,Y 427.267,Z 449.761,A -85,B 0,C 180,E1 -9705.886,E2 -9705.886} C_VEL
LIN {X 0,Y 426.794,Z 460.566,A -85,B 0,C 180,E1 -9706.792,E2 -9706.792} C_VEL
LIN {X 0,Y 426.279,Z 470.908,A -85,B 0,C 180,E1 -9707.865,E2 -9707.865} C_VEL
LIN {X 0,Y 425.705,Z 480.219,A -85,B 0,C 180,E1 -9709.056,E2 -9709.056} C_VEL
LIN {X 0,Y 425.247,Z 489.31,A -85,B 0,C 180,E1 -9710.487,E2 -9710.487} C_VEL
LIN {X 0,Y 424.849,Z 496.556,A -85,B 0,C 180,E1 -9711.917,E2 -9711.917} C_VEL
LIN {X 0,Y 424.632,Z 502.337,A -85,B 0,C 180,E1 -9713.347,E2 -9713.347} C_VEL
LIN {X 0,Y 424.406,Z 506.864,A -85,B 0,C 180,E1 -9714.774,E2 -9714.774} C_VEL
LIN {X 0,Y 424.361,Z 510.263,A -85,B 0,C 180,E1 -9716.202,E2 -9716.202} C_VEL
LIN {X 0,Y 424.321,Z 511.96,A -85,B 0,C 180,E1 -9717.152,E2 -9717.152} C_VEL
LIN {X 0,Y 424.201,Z 513.228,A -85,B 0,C 180,E1 -9718.101,E2 -9718.101} C_VEL
LIN {X 0,Y 424.144,Z 514.028,A -85,B 0,C 180,E1 -9719.051,E2 -9719.051} C_VEL
LIN {X 0,Y 424.142,Z 514.422,A -85,B 0,C 180,E1 -9720,E2 -9720} C_VEL
LIN {X 0,Y 424.171,Z 514.411,A -85,B 0,C 180,E1 -9720.949,E2 -9720.949} C_VEL
LIN {X 0,Y 424.233,Z 513.947,A -85,B 0,C 180,E1 -9721.899,E2 -9721.899} C_VEL
LIN {X 0,Y 424.334,Z 513.049,A -85,B 0,C 180,E1 -9722.848,E2 -9722.848} C_VEL
LIN {X 0,Y 424.469,Z 511.739,A -85,B 0,C 180,E1 -9723.797,E2 -9723.797} C_VEL
LIN {X 0,Y 424.441,Z 508.938,A -85,B 0,C 180,E1 -9725.225,E2 -9725.225} C_VEL
LIN {X 0,Y 424.836,Z 505.045,A -85,B 0,C 180,E1 -9726.65,E2 -9726.65} C_VEL
LIN {X 0,Y 425.072,Z 499.998,A -85,B 0,C 180,E1 -9728.079,E2 -9728.079} C_VEL
LIN {X 0,Y 425.558,Z 493.584,A -85,B 0,C 180,E1 -9729.506,E2 -9729.506} C_VEL
LIN {X 0,Y 426.108,Z 485.546,A -85,B 0,C 180,E1 -9730.934,E2 -9730.934} C_VEL
LIN {X 0,Y 426.595,Z 477.353,A -85,B 0,C 180,E1 -9732.125,E2 -9732.125} C_VEL
LIN {X 0,Y 427.298,Z 467.327,A -85,B 0,C 180,E1 -9733.313,E2 -9733.313} C_VEL
LIN {X 0,Y 427.998,Z 456.448,A -85,B 0,C 180,E1 -9734.344,E2 -9734.344} C_VEL
LIN {X 0,Y 428.634,Z 445.052,A -85,B 0,C 180,E1 -9735.209,E2 -9735.209} C_VEL
LIN {X 0,Y 429.187,Z 432.957,A -85,B 0,C 180,E1 -9735.919,E2 -9735.919} C_VEL
LIN {X 0,Y 429.664,Z 419.773,A -85,B 0,C 180,E1 -9736.481,E2 -9736.481} C_VEL
LIN {X 0,Y 429.99,Z 405.983,A -85,B 0,C 180,E1 -9736.865,E2 -9736.865} C_VEL
LIN {X 0,Y 432.073,Z 327.273,A -85,B 0,C 180,E1 -9738.612,E2 -9738.612} C_VEL
LIN {X 0,Y 432.004,Z 322.283,A -85,B 0,C 180,E1 -9738.741,E2 -9738.741} C_VEL
LIN {X 0,Y 428.61,Z 309.204,A -85,B 0,C 180,E1 -9739.3,E2 -9739.3} C_VEL
LIN {X 0,Y 428.031,Z 307.248,A -85,B 0,C 180,E1 -9739.42,E2 -9739.42} C_VEL
LIN {X 0,Y 427.539,Z 302.653,A -85,B 0,C 180,E1 -9740.75,E2 -9740.75} C_VEL
LIN {X 0,Y 425.75,Z 294.481,A -85,B 0,C 180,E1 -9743.339,E2 -9743.339} C_VEL
LIN {X 0,Y 425.322,Z 292.509,A -85,B 0,C 180,E1 -9744.01,E2 -9744.01} C_VEL
LIN {X 0,Y 425.241,Z 292.518,A -85,B 0,C 180,E1 -9747.565,E2 -9747.565} C_VEL
LIN {X 0,Y 425.288,Z 292.511,A -85,B 0,C 180,E1 -9750.759,E2 -9750.759} C_VEL
LIN {X 0,Y 425.291,Z 292.509,A -85,B 0,C 180,E1 -9754.283,E2 -9754.283} C_VEL
LIN {X 0,Y 425.272,Z 292.511,A -85,B 0,C 180,E1 -9757.695,E2 -9757.695} C_VEL
LIN {X 0,Y 425.246,Z 292.516,A -85,B 0,C 180,E1 -9760.514,E2 -9760.514} C_VEL
LIN {X 0,Y 425.248,Z 292.515,A -85,B 0,C 180,E1 -9763.348,E2 -9763.348} C_VEL
LIN {X 0,Y 425.258,Z 292.513,A -85,B 0,C 180,E1 -9766.043,E2 -9766.043} C_VEL
LIN {X 0,Y 425.251,Z 292.515,A -85,B 0,C 180,E1 -9768.618,E2 -9768.618} C_VEL
LIN {X 0,Y 425.281,Z 292.51,A -85,B 0,C 180,E1 -9771.099,E2 -9771.099} C_VEL
LIN {X 0,Y 425.302,Z 292.509,A -85,B 0,C 180,E1 -9774.663,E2 -9774.663} C_VEL
LIN {X 0,Y 425.269,Z 292.519,A -85,B 0,C 180,E1 -9778.073,E2 -9778.073} C_VEL
LIN {X 0,Y 425.312,Z 292.618,A -85,B 0,C 180,E1 -9780.309,E2 -9780.309} C_VEL
LIN {X 0,Y 427.686,Z 302.039,A -85,B 0,C 180,E1 -9782.813,E2 -9782.813} C_VEL
LIN {X 0,Y 429.238,Z 310.349,A -85,B 0,C 180,E1 -9784.804,E2 -9784.804} C_VEL
LIN {X 0,Y 428.689,Z 317.858,A -85,B 0,C 180,E1 -9786.369,E2 -9786.369} C_VEL
LIN {X 0,Y 427.552,Z 331.37,A -85,B 0,C 180,E1 -9789.076,E2 -9789.076} C_VEL
LIN {X 0,Y 427.032,Z 339.155,A -85,B 0,C 180,E1 -9790.563,E2 -9790.563} C_VEL
LIN {X 0,Y 430.099,Z 356.001,A -85,B 0,C 180,E1 -9791.181,E2 -9791.181} C_VEL
LIN {X 0,Y 431.39,Z 368.556,A -85,B 0,C 180,E1 -9791.567,E2 -9791.567} C_VEL
LIN {X 0,Y 429.399,Z 450.694,A -85,B 0,C 180,E1 -9793.386,E2 -9793.386} C_VEL
LIN {X 0,Y 428.78,Z 464.476,A -85,B 0,C 180,E1 -9793.881,E2 -9793.881} C_VEL
LIN {X 0,Y 428.066,Z 476.959,A -85,B 0,C 180,E1 -9794.526,E2 -9794.526} C_VEL
LIN {X 0,Y 427.375,Z 489.19,A -85,B 0,C 180,E1 -9795.354,E2 -9795.354} C_VEL
LIN {X 0,Y 426.706,Z 499.514,A -85,B 0,C 180,E1 -9796.231,E2 -9796.231} C_VEL
LIN {X 0,Y 426.004,Z 510.336,A -85,B 0,C 180,E1 -9797.373,E2 -9797.373} C_VEL
LIN {X 0,Y 425.488,Z 519.57,A -85,B 0,C 180,E1 -9798.567,E2 -9798.567} C_VEL
LIN {X 0,Y 424.921,Z 528.61,A -85,B 0,C 180,E1 -9799.998,E2 -9799.998} C_VEL
LIN {X 0,Y 424.539,Z 535.833,A -85,B 0,C 180,E1 -9801.431,E2 -9801.431} C_VEL
LIN {X 0,Y 424.327,Z 541.633,A -85,B 0,C 180,E1 -9802.863,E2 -9802.863} C_VEL
LIN {X 0,Y 424.194,Z 546.185,A -85,B 0,C 180,E1 -9804.294,E2 -9804.294} C_VEL
LIN {X 0,Y 424.209,Z 548.61,A -85,B 0,C 180,E1 -9805.247,E2 -9805.247} C_VEL
LIN {X 0,Y 424.11,Z 550.523,A -85,B 0,C 180,E1 -9806.198,E2 -9806.198} C_VEL
LIN {X 0,Y 424.176,Z 551.983,A -85,B 0,C 180,E1 -9807.15,E2 -9807.15} C_VEL
LIN {X 0,Y 424.165,Z 553.019,A -85,B 0,C 180,E1 -9808.1,E2 -9808.1} C_VEL
LIN {X 0,Y 424.137,Z 553.625,A -85,B 0,C 180,E1 -9809.05,E2 -9809.05} C_VEL
LIN {X 0,Y 424.149,Z 553.762,A -85,B 0,C 180,E1 -9809.999,E2 -9809.999} C_VEL
LIN {X 0,Y 424.137,Z 553.481,A -85,B 0,C 180,E1 -9810.948,E2 -9810.948} C_VEL
LIN {X 0,Y 424.166,Z 552.787,A -85,B 0,C 180,E1 -9811.898,E2 -9811.898} C_VEL
LIN {X 0,Y 424.212,Z 551.63,A -85,B 0,C 180,E1 -9812.848,E2 -9812.848} C_VEL
LIN {X 0,Y 424.151,Z 549.051,A -85,B 0,C 180,E1 -9814.275,E2 -9814.275} C_VEL
LIN {X 0,Y 424.194,Z 545.394,A -85,B 0,C 180,E1 -9815.704,E2 -9815.704} C_VEL
LIN {X 0,Y 424.338,Z 540.557,A -85,B 0,C 180,E1 -9817.135,E2 -9817.135} C_VEL
LIN {X 0,Y 424.553,Z 533.296,A -85,B 0,C 180,E1 -9818.807,E2 -9818.807} C_VEL
LIN {X 0,Y 424.882,Z 525.898,A -85,B 0,C 180,E1 -9820.242,E2 -9820.242} C_VEL
LIN {X 0,Y 425.361,Z 518.36,A -85,B 0,C 180,E1 -9821.435,E2 -9821.435} C_VEL
LIN {X 0,Y 425.919,Z 509.207,A -85,B 0,C 180,E1 -9822.628,E2 -9822.628} C_VEL
LIN {X 0,Y 426.592,Z 499.133,A -85,B 0,C 180,E1 -9823.686,E2 -9823.686} C_VEL
LIN {X 0,Y 427.257,Z 487.659,A -85,B 0,C 180,E1 -9824.648,E2 -9824.648} C_VEL
LIN {X 0,Y 427.902,Z 475.837,A -85,B 0,C 180,E1 -9825.418,E2 -9825.418} C_VEL
LIN {X 0,Y 428.465,Z 463.457,A -85,B 0,C 180,E1 -9826.007,E2 -9826.007} C_VEL
LIN {X 0,Y 428.967,Z 450.769,A -85,B 0,C 180,E1 -9826.415,E2 -9826.415} C_VEL
LIN {X 0,Y 429.344,Z 422.42,A -85,B 0,C 180,E1 -9826.921,E2 -9826.921} C_VEL
LIN {X 0,Y 429.816,Z 366.044,A -85,B 0,C 180,E1 -9827.862,E2 -9827.862} C_VEL
LIN {X 0,Y 426.421,Z 341.962,A -85,B 0,C 180,E1 -9828.45,E2 -9828.45} C_VEL
LIN {X 0,Y 427.485,Z 323.05,A -85,B 0,C 180,E1 -9831.962,E2 -9831.962} C_VEL
LIN {X 0,Y 428.407,Z 308.373,A -85,B 0,C 180,E1 -9834.728,E2 -9834.728} C_VEL
LIN {X 0,Y 426.577,Z 298.435,A -85,B 0,C 180,E1 -9836.74,E2 -9836.74} C_VEL
LIN {X 0,Y 425.375,Z 292.501,A -85,B 0,C 180,E1 -9838.023,E2 -9838.023} C_VEL
LIN {X 0,Y 425.285,Z 292.507,A -85,B 0,C 180,E1 -9840.815,E2 -9840.815} C_VEL
LIN {X 0,Y 425.308,Z 292.507,A -85,B 0,C 180,E1 -9844.287,E2 -9844.287} C_VEL
LIN {X 0,Y 425.272,Z 292.512,A -85,B 0,C 180,E1 -9847.693,E2 -9847.693} C_VEL
LIN {X 0,Y 425.271,Z 292.509,A -85,B 0,C 180,E1 -9850.519,E2 -9850.519} C_VEL
LIN {X 0,Y 425.256,Z 292.515,A -85,B 0,C 180,E1 -9853.955,E2 -9853.955} C_VEL
LIN {X 0,Y 425.263,Z 292.511,A -85,B 0,C 180,E1 -9857.345,E2 -9857.345} C_VEL
LIN {X 0,Y 425.274,Z 292.509,A -85,B 0,C 180,E1 -9861.099,E2 -9861.099} C_VEL
LIN {X 0,Y 425.291,Z 292.506,A -85,B 0,C 180,E1 -9864.663,E2 -9864.663} C_VEL
LIN {X 0,Y 425.256,Z 292.512,A -85,B 0,C 180,E1 -9868.072,E2 -9868.072} C_VEL
LIN {X 0,Y 425.296,Z 292.51,A -85,B 0,C 180,E1 -9871.365,E2 -9871.365} C_VEL
LIN {X 0,Y 425.255,Z 292.511,A -85,B 0,C 180,E1 -9874.552,E2 -9874.552} C_VEL
LIN {X 0,Y 425.27,Z 292.509,A -85,B 0,C 180,E1 -9876.633,E2 -9876.633} C_VEL
LIN {X 0,Y 425.286,Z 292.51,A -85,B 0,C 180,E1 -9879.694,E2 -9879.694} C_VEL
LIN {X 0,Y 425.323,Z 292.503,A -85,B 0,C 180,E1 -9882.697,E2 -9882.697} C_VEL
LIN {X 0,Y 425.332,Z 292.504,A -85,B 0,C 180,E1 -9885.649,E2 -9885.649} C_VEL
LIN {X 0,Y 425.337,Z 292.502,A -85,B 0,C 180,E1 -9888.564,E2 -9888.564} C_VEL
LIN {X 0,Y 425.398,Z 292.496,A -85,B 0,C 180,E1 -9891.449,E2 -9891.449} C_VEL
LIN {X 0,Y 425.493,Z 292.482,A -85,B 0,C 180,E1 -9894.312,E2 -9894.312} C_VEL
LIN {X 0,Y 425.558,Z 292.474,A -85,B 0,C 180,E1 -9898.107,E2 -9898.107} C_VEL
LIN {X 0,Y 425.498,Z 292.485,A -85,B 0,C 180,E1 -9900.946,E2 -9900.946} C_VEL
LIN {X 0,Y 425.5,Z 292.485,A -85,B 0,C 180,E1 -9902.84,E2 -9902.84} C_VEL
LIN {X 0,Y 425.465,Z 292.488,A -85,B 0,C 180,E1 -9906.604,E2 -9906.604} C_VEL
LIN {X 0,Y 425.384,Z 292.497,A -85,B 0,C 180,E1 -9909.51,E2 -9909.51} C_VEL
LIN {X 0,Y 425.385,Z 292.498,A -85,B 0,C 180,E1 -9912.904,E2 -9912.904} C_VEL
LIN {X 0,Y 425.352,Z 292.503,A -85,B 0,C 180,E1 -9916.605,E2 -9916.605} C_VEL
LIN {X 0,Y 425.32,Z 292.504,A -85,B 0,C 180,E1 -9919.636,E2 -9919.636} C_VEL
LIN {X 0,Y 425.28,Z 292.511,A -85,B 0,C 180,E1 -9922.339,E2 -9922.339} C_VEL
LIN {X 0,Y 425.311,Z 292.507,A -85,B 0,C 180,E1 -9924.657,E2 -9924.657} C_VEL
LIN {X 0,Y 425.29,Z 292.508,A -85,B 0,C 180,E1 -9927.562,E2 -9927.562} C_VEL
LIN {X 0,Y 425.28,Z 292.511,A -85,B 0,C 180,E1 -9930.817,E2 -9930.817} C_VEL
LIN {X 0,Y 425.304,Z 292.509,A -85,B 0,C 180,E1 -9934.289,E2 -9934.289} C_VEL
LIN {X 0,Y 425.27,Z 292.51,A -85,B 0,C 180,E1 -9937.695,E2 -9937.695} C_VEL
LIN {X 0,Y 425.27,Z 292.512,A -85,B 0,C 180,E1 -9940.521,E2 -9940.521} C_VEL
LIN {X 0,Y 425.255,Z 292.514,A -85,B 0,C 180,E1 -9943.957,E2 -9943.957} C_VEL
LIN {X 0,Y 425.27,Z 292.51,A -85,B 0,C 180,E1 -9947.348,E2 -9947.348} C_VEL
LIN {X 0,Y 425.282,Z 292.511,A -85,B 0,C 180,E1 -9949.874,E2 -9949.874} C_VEL
LIN {X 0,Y 425.274,Z 292.513,A -85,B 0,C 180,E1 -9952.49,E2 -9952.49} C_VEL
LIN {X 0,Y 425.302,Z 292.508,A -85,B 0,C 180,E1 -9955.818,E2 -9955.818} C_VEL
LIN {X 0,Y 425.288,Z 292.508,A -85,B 0,C 180,E1 -9959.24,E2 -9959.24} C_VEL
LIN {X 0,Y 425.347,Z 292.504,A -85,B 0,C 180,E1 -9962.443,E2 -9962.443} C_VEL
LIN {X 0,Y 425.348,Z 292.502,A -85,B 0,C 180,E1 -9965.603,E2 -9965.603} C_VEL
LIN {X 0,Y 425.293,Z 292.51,A -85,B 0,C 180,E1 -9968.683,E2 -9968.683} C_VEL
LIN {X 0,Y 425.358,Z 292.526,A -85,B 0,C 180,E1 -9970.911,E2 -9970.911} C_VEL
LIN {X 0,Y 426.57,Z 296.581,A -85,B 0,C 180,E1 -9971.233,E2 -9971.233} C_VEL
LIN {X 0,Y 427.823,Z 301.295,A -85,B 0,C 180,E1 -9971.373,E2 -9971.373} C_VEL
LIN {X 0,Y 430.777,Z 321.777,A -85,B 0,C 180,E1 -9971.862,E2 -9971.862} C_VEL
LIN {X 0,Y 429.773,Z 410.5,A -85,B 0,C 180,E1 -9973.372,E2 -9973.372} C_VEL
LIN {X 0,Y 429.48,Z 424.073,A -85,B 0,C 180,E1 -9973.788,E2 -9973.788} C_VEL
LIN {X 0,Y 428.933,Z 436.668,A -85,B 0,C 180,E1 -9974.377,E2 -9974.377} C_VEL
LIN {X 0,Y 428.362,Z 448.788,A -85,B 0,C 180,E1 -9975.148,E2 -9975.148} C_VEL
LIN {X 0,Y 427.844,Z 458.471,A -85,B 0,C 180,E1 -9975.934,E2 -9975.934} C_VEL
LIN {X 0,Y 427.235,Z 468.434,A -85,B 0,C 180,E1 -9976.928,E2 -9976.928} C_VEL
LIN {X 0,Y 426.512,Z 478.049,A -85,B 0,C 180,E1 -9978.115,E2 -9978.115} C_VEL
LIN {X 0,Y 426.46,Z 478.857,A -85,B 0,C 180,E1 -9978.226,E2 -9978.226} C_VEL
LIN {X 0,Y 425.536,Z 482.916,A -85,B 0,C 180,E1 -9978.793,E2 -9978.793} C_VEL
LIN {X 0,Y 422.242,Z 489.179,A -85,B 0,C 180,E1 -9979.736,E2 -9979.736} C_VEL
LIN {X 0,Y 418.962,Z 494.797,A -85,B 0,C 180,E1 -9980.759,E2 -9980.759} C_VEL
LIN {X 0,Y 418.076,Z 497.841,A -85,B 0,C 180,E1 -9981.443,E2 -9981.443} C_VEL
LIN {X 0,Y 417.698,Z 503.827,A -85,B 0,C 180,E1 -9983.079,E2 -9983.079} C_VEL
LIN {X 0,Y 417.369,Z 508.297,A -85,B 0,C 180,E1 -9984.687,E2 -9984.687} C_VEL
LIN {X 0,Y 417.323,Z 511.21,A -85,B 0,C 180,E1 -9986.138,E2 -9986.138} C_VEL
LIN {X 0,Y 417.26,Z 512.627,A -85,B 0,C 180,E1 -9987.105,E2 -9987.105} C_VEL
LIN {X 0,Y 417.063,Z 514.238,A -85,B 0,C 180,E1 -9989.035,E2 -9989.035} C_VEL
LIN {X 0,Y 417.056,Z 514.472,A -85,B 0,C 180,E1 -9990.001,E2 -9990.001} C_VEL
LIN {X 0,Y 417.128,Z 513.699,A -85,B 0,C 180,E1 -9991.932,E2 -9991.932} C_VEL
LIN {X 0,Y 417.259,Z 512.734,A -85,B 0,C 180,E1 -9992.897,E2 -9992.897} C_VEL
LIN {X 0,Y 417.316,Z 511.376,A -85,B 0,C 180,E1 -9993.864,E2 -9993.864} C_VEL
LIN {X 0,Y 417.367,Z 508.523,A -85,B 0,C 180,E1 -9995.315,E2 -9995.315} C_VEL
LIN {X 0,Y 417.685,Z 504.182,A -85,B 0,C 180,E1 -9996.907,E2 -9996.907} C_VEL
LIN {X 0,Y 417.961,Z 499.607,A -85,B 0,C 180,E1 -9998.218,E2 -9998.218} C_VEL
LIN {X 0,Y 418.469,Z 493.26,A -85,B 0,C 180,E1 -9999.669,E2 -9999.669} C_VEL
LIN {X 0,Y 419.051,Z 485.365,A -85,B 0,C 180,E1 -10001.121,E2 -10001.121} C_VEL
LIN {X 0,Y 419.682,Z 477.289,A -85,B 0,C 180,E1 -10002.329,E2 -10002.329} C_VEL
LIN {X 0,Y 420.5,Z 467.372,A -85,B 0,C 180,E1 -10003.533,E2 -10003.533} C_VEL
LIN {X 0,Y 421.125,Z 456.235,A -85,B 0,C 180,E1 -10004.621,E2 -10004.621} C_VEL
LIN {X 0,Y 421.764,Z 445.314,A -85,B 0,C 180,E1 -10005.464,E2 -10005.464} C_VEL
LIN {X 0,Y 422.32,Z 433.027,A -85,B 0,C 180,E1 -10006.186,E2 -10006.186} C_VEL
LIN {X 0,Y 422.831,Z 420.25,A -85,B 0,C 180,E1 -10006.725,E2 -10006.725} C_VEL
LIN {X 0,Y 423.087,Z 408.197,A -85,B 0,C 180,E1 -10007.056,E2 -10007.056} C_VEL
LIN {X 0,Y 423.984,Z 321.214,A -85,B 0,C 180,E1 -10008.55,E2 -10008.55} C_VEL
LIN {X 0,Y 420.611,Z 300.336,A -85,B 0,C 180,E1 -10009.077,E2 -10009.077} C_VEL
LIN {X 0,Y 419.114,Z 296.191,A -85,B 0,C 180,E1 -10009.235,E2 -10009.235} C_VEL
LIN {X 0,Y 418.337,Z 293.378,A -85,B 0,C 180,E1 -10009.473,E2 -10009.473} C_VEL
LIN {X 0,Y 418.242,Z 293.385,A -85,B 0,C 180,E1 -10012.737,E2 -10012.737} C_VEL
LIN {X 0,Y 418.273,Z 293.385,A -85,B 0,C 180,E1 -10015.905,E2 -10015.905} C_VEL
LIN {X 0,Y 418.27,Z 293.382,A -85,B 0,C 180,E1 -10019.162,E2 -10019.162} C_VEL
LIN {X 0,Y 418.262,Z 293.382,A -85,B 0,C 180,E1 -10022.844,E2 -10022.844} C_VEL
LIN {X 0,Y 418.249,Z 293.384,A -85,B 0,C 180,E1 -10026.238,E2 -10026.238} C_VEL
LIN {X 0,Y 418.256,Z 293.386,A -85,B 0,C 180,E1 -10029.682,E2 -10029.682} C_VEL
LIN {X 0,Y 418.237,Z 293.385,A -85,B 0,C 180,E1 -10032.322,E2 -10032.322} C_VEL
LIN {X 0,Y 418.243,Z 293.388,A -85,B 0,C 180,E1 -10035.109,E2 -10035.109} C_VEL
LIN {X 0,Y 418.245,Z 293.385,A -85,B 0,C 180,E1 -10037.767,E2 -10037.767} C_VEL
LIN {X 0,Y 418.258,Z 293.383,A -85,B 0,C 180,E1 -10040.62,E2 -10040.62} C_VEL
LIN {X 0,Y 418.248,Z 293.383,A -85,B 0,C 180,E1 -10043.976,E2 -10043.976} C_VEL
LIN {X 0,Y 418.263,Z 293.385,A -85,B 0,C 180,E1 -10047.156,E2 -10047.156} C_VEL
LIN {X 0,Y 418.274,Z 293.386,A -85,B 0,C 180,E1 -10050.896,E2 -10050.896} C_VEL
LIN {X 0,Y 418.267,Z 293.381,A -85,B 0,C 180,E1 -10054.096,E2 -10054.096} C_VEL
LIN {X 0,Y 418.243,Z 293.385,A -85,B 0,C 180,E1 -10057.264,E2 -10057.264} C_VEL
LIN {X 0,Y 418.343,Z 293.582,A -85,B 0,C 180,E1 -10058.826,E2 -10058.826} C_VEL
LIN {X 0,Y 419.659,Z 301.934,A -85,B 0,C 180,E1 -10060.939,E2 -10060.939} C_VEL
LIN {X 0,Y 419.625,Z 304.063,A -85,B 0,C 180,E1 -10061.429,E2 -10061.429} C_VEL
LIN {X 0,Y 423.17,Z 323.364,A -85,B 0,C 180,E1 -10061.971,E2 -10061.971} C_VEL
LIN {X 0,Y 421.571,Z 412.091,A -85,B 0,C 180,E1 -10063.816,E2 -10063.816} C_VEL
LIN {X 0,Y 421.28,Z 425.791,A -85,B 0,C 180,E1 -10064.302,E2 -10064.302} C_VEL
LIN {X 0,Y 420.721,Z 438.219,A -85,B 0,C 180,E1 -10064.932,E2 -10064.932} C_VEL
LIN {X 0,Y 420.277,Z 450.292,A -85,B 0,C 180,E1 -10065.752,E2 -10065.752} C_VEL
LIN {X 0,Y 419.764,Z 461.259,A -85,B 0,C 180,E1 -10066.69,E2 -10066.69} C_VEL
LIN {X 0,Y 419.222,Z 471.518,A -85,B 0,C 180,E1 -10067.781,E2 -10067.781} C_VEL
LIN {X 0,Y 418.626,Z 481.633,A -85,B 0,C 180,E1 -10069.113,E2 -10069.113} C_VEL
LIN {X 0,Y 418.207,Z 489.156,A -85,B 0,C 180,E1 -10070.325,E2 -10070.325} C_VEL
LIN {X 0,Y 417.816,Z 496.536,A -85,B 0,C 180,E1 -10071.78,E2 -10071.78} C_VEL
LIN {X 0,Y 417.564,Z 502.395,A -85,B 0,C 180,E1 -10073.234,E2 -10073.234} C_VEL
LIN {X 0,Y 417.349,Z 506.995,A -85,B 0,C 180,E1 -10074.686,E2 -10074.686} C_VEL
LIN {X 0,Y 417.266,Z 510.461,A -85,B 0,C 180,E1 -10076.137,E2 -10076.137} C_VEL
LIN {X 0,Y 417.255,Z 512.191,A -85,B 0,C 180,E1 -10077.104,E2 -10077.104} C_VEL
LIN {X 0,Y 417.129,Z 513.501,A -85,B 0,C 180,E1 -10078.069,E2 -10078.069} C_VEL
LIN {X 0,Y 417.064,Z 514.339,A -85,B 0,C 180,E1 -10079.034,E2 -10079.034} C_VEL
LIN {X 0,Y 417.059,Z 514.759,A -85,B 0,C 180,E1 -10080,E2 -10080} C_VEL
LIN {X 0,Y 417.09,Z 514.772,A -85,B 0,C 180,E1 -10080.965,E2 -10080.965} C_VEL
LIN {X 0,Y 417.158,Z 514.352,A -85,B 0,C 180,E1 -10081.931,E2 -10081.931} C_VEL
LIN {X 0,Y 417.272,Z 513.476,A -85,B 0,C 180,E1 -10082.896,E2 -10082.896} C_VEL
LIN {X 0,Y 417.411,Z 512.189,A -85,B 0,C 180,E1 -10083.862,E2 -10083.862} C_VEL
LIN {X 0,Y 417.388,Z 509.429,A -85,B 0,C 180,E1 -10085.314,E2 -10085.314} C_VEL
LIN {X 0,Y 417.799,Z 505.575,A -85,B 0,C 180,E1 -10086.762,E2 -10086.762} C_VEL
LIN {X 0,Y 418.063,Z 500.576,A -85,B 0,C 180,E1 -10088.215,E2 -10088.215} C_VEL
LIN {X 0,Y 418.601,Z 494.232,A -85,B 0,C 180,E1 -10089.665,E2 -10089.665} C_VEL
LIN {X 0,Y 419.174,Z 486.248,A -85,B 0,C 180,E1 -10091.117,E2 -10091.117} C_VEL
LIN {X 0,Y 419.697,Z 478.132,A -85,B 0,C 180,E1 -10092.328,E2 -10092.328} C_VEL
LIN {X 0,Y 420.448,Z 468.218,A -85,B 0,C 180,E1 -10093.534,E2 -10093.534} C_VEL
LIN {X 0,Y 421.193,Z 457.478,A -85,B 0,C 180,E1 -10094.581,E2 -10094.581} C_VEL
LIN {X 0,Y 421.87,Z 446.263,A -85,B 0,C 180,E1 -10095.459,E2 -10095.459} C_VEL
LIN {X 0,Y 422.521,Z 433.357,A -85,B 0,C 180,E1 -10096.239,E2 -10096.239} C_VEL
LIN {X 0,Y 423.017,Z 420.291,A -85,B 0,C 180,E1 -10096.809,E2 -10096.809} C_VEL
LIN {X 0,Y 423.389,Z 406.741,A -85,B 0,C 180,E1 -10097.198,E2 -10097.198} C_VEL
LIN {X 0,Y 425.688,Z 327.578,A -85,B 0,C 180,E1 -10099.017,E2 -10099.017} C_VEL
LIN {X 0,Y 425.478,Z 322.959,A -85,B 0,C 180,E1 -10099.151,E2 -10099.151} C_VEL
LIN {X 0,Y 422.236,Z 310.842,A -85,B 0,C 180,E1 -10099.704,E2 -10099.704} C_VEL
LIN {X 0,Y 421.159,Z 307.813,A -85,B 0,C 180,E1 -10099.89,E2 -10099.89} C_VEL
LIN {X 0,Y 420.25,Z 302.279,A -85,B 0,C 180,E1 -10101.587,E2 -10101.587} C_VEL
LIN {X 0,Y 418.261,Z 293.388,A -85,B 0,C 180,E1 -10104.574,E2 -10104.574} C_VEL
LIN {X 0,Y 418.203,Z 293.394,A -85,B 0,C 180,E1 -10108.07,E2 -10108.07} C_VEL
LIN {X 0,Y 418.236,Z 293.39,A -85,B 0,C 180,E1 -10111.018,E2 -10111.018} C_VEL
LIN {X 0,Y 418.23,Z 293.389,A -85,B 0,C 180,E1 -10113.679,E2 -10113.679} C_VEL
LIN {X 0,Y 418.235,Z 293.389,A -85,B 0,C 180,E1 -10117.225,E2 -10117.225} C_VEL
LIN {X 0,Y 418.21,Z 293.392,A -85,B 0,C 180,E1 -10120.867,E2 -10120.867} C_VEL
LIN {X 0,Y 418.204,Z 293.392,A -85,B 0,C 180,E1 -10123.728,E2 -10123.728} C_VEL
LIN {X 0,Y 418.201,Z 293.395,A -85,B 0,C 180,E1 -10126.447,E2 -10126.447} C_VEL
LIN {X 0,Y 418.21,Z 293.392,A -85,B 0,C 180,E1 -10129.133,E2 -10129.133} C_VEL
LIN {X 0,Y 418.24,Z 293.39,A -85,B 0,C 180,E1 -10132.775,E2 -10132.775} C_VEL
LIN {X 0,Y 418.252,Z 293.389,A -85,B 0,C 180,E1 -10136.322,E2 -10136.322} C_VEL
LIN {X 0,Y 418.277,Z 293.549,A -85,B 0,C 180,E1 -10139.73,E2 -10139.73} C_VEL
LIN {X 0,Y 420.678,Z 302.738,A -85,B 0,C 180,E1 -10142.306,E2 -10142.306} C_VEL
LIN {X 0,Y 422.448,Z 312.1,A -85,B 0,C 180,E1 -10144.634,E2 -10144.634} C_VEL
LIN {X 0,Y 421.996,Z 318.287,A -85,B 0,C 180,E1 -10145.97,E2 -10145.97} C_VEL
LIN {X 0,Y 420.649,Z 332.781,A -85,B 0,C 180,E1 -10148.948,E2 -10148.948} C_VEL
LIN {X 0,Y 420.215,Z 338.465,A -85,B 0,C 180,E1 -10150.081,E2 -10150.081} C_VEL
LIN {X 0,Y 423.458,Z 355.731,A -85,B 0,C 180,E1 -10150.757,E2 -10150.757} C_VEL
LIN {X 0,Y 424.908,Z 368.712,A -85,B 0,C 180,E1 -10151.183,E2 -10151.183} C_VEL
LIN {X 0,Y 422.743,Z 450.392,A -85,B 0,C 180,E1 -10153.054,E2 -10153.054} C_VEL
LIN {X 0,Y 422.07,Z 464.037,A -85,B 0,C 180,E1 -10153.556,E2 -10153.556} C_VEL
LIN {X 0,Y 421.259,Z 477.464,A -85,B 0,C 180,E1 -10154.269,E2 -10154.269} C_VEL
LIN {X 0,Y 420.526,Z 489.484,A -85,B 0,C 180,E1 -10155.11,E2 -10155.11} C_VEL
LIN {X 0,Y 419.74,Z 500.633,A -85,B 0,C 180,E1 -10156.1,E2 -10156.1} C_VEL
LIN {X 0,Y 419.054,Z 510.372,A -85,B 0,C 180,E1 -10157.163,E2 -10157.163} C_VEL
LIN {X 0,Y 418.513,Z 519.521,A -85,B 0,C 180,E1 -10158.374,E2 -10158.374} C_VEL
LIN {X 0,Y 417.931,Z 527.113,A -85,B 0,C 180,E1 -10159.584,E2 -10159.584} C_VEL
LIN {X 0,Y 417.544,Z 534.596,A -85,B 0,C 180,E1 -10161.042,E2 -10161.042} C_VEL
LIN {X 0,Y 417.324,Z 539.679,A -85,B 0,C 180,E1 -10162.256,E2 -10162.256} C_VEL
LIN {X 0,Y 417.142,Z 544.685,A -85,B 0,C 180,E1 -10163.739,E2 -10163.739} C_VEL
LIN {X 0,Y 417.116,Z 548.362,A -85,B 0,C 180,E1 -10165.166,E2 -10165.166} C_VEL
LIN {X 0,Y 417.025,Z 550.246,A -85,B 0,C 180,E1 -10166.134,E2 -10166.134} C_VEL
LIN {X 0,Y 417.072,Z 551.693,A -85,B 0,C 180,E1 -10167.101,E2 -10167.101} C_VEL
LIN {X 0,Y 417.091,Z 552.718,A -85,B 0,C 180,E1 -10168.068,E2 -10168.068} C_VEL
LIN {X 0,Y 417.056,Z 553.289,A -85,B 0,C 180,E1 -10169.033,E2 -10169.033} C_VEL
LIN {X 0,Y 417.065,Z 553.407,A -85,B 0,C 180,E1 -10169.999,E2 -10169.999} C_VEL
LIN {X 0,Y 417.056,Z 553.108,A -85,B 0,C 180,E1 -10170.965,E2 -10170.965} C_VEL
LIN {X 0,Y 417.093,Z 552.391,A -85,B 0,C 180,E1 -10171.93,E2 -10171.93} C_VEL
LIN {X 0,Y 417.125,Z 551.192,A -85,B 0,C 180,E1 -10172.896,E2 -10172.896} C_VEL
LIN {X 0,Y 417.077,Z 548.563,A -85,B 0,C 180,E1 -10174.348,E2 -10174.348} C_VEL
LIN {X 0,Y 417.112,Z 544.849,A -85,B 0,C 180,E1 -10175.801,E2 -10175.801} C_VEL
LIN {X 0,Y 417.262,Z 539.952,A -85,B 0,C 180,E1 -10177.256,E2 -10177.256} C_VEL
LIN {X 0,Y 417.56,Z 531.853,A -85,B 0,C 180,E1 -10179.2,E2 -10179.2} C_VEL
LIN {X 0,Y 417.945,Z 524.214,A -85,B 0,C 180,E1 -10180.658,E2 -10180.658} C_VEL
LIN {X 0,Y 418.528,Z 516.377,A -85,B 0,C 180,E1 -10181.87,E2 -10181.87} C_VEL
LIN {X 0,Y 419.13,Z 506.93,A -85,B 0,C 180,E1 -10183.065,E2 -10183.065} C_VEL
LIN {X 0,Y 419.843,Z 496.119,A -85,B 0,C 180,E1 -10184.17,E2 -10184.17} C_VEL
LIN {X 0,Y 420.443,Z 485.769,A -85,B 0,C 180,E1 -10185.015,E2 -10185.015} C_VEL
LIN {X 0,Y 421.2,Z 473.315,A -85,B 0,C 180,E1 -10185.793,E2 -10185.793} C_VEL
LIN {X 0,Y 421.761,Z 460.92,A -85,B 0,C 180,E1 -10186.362,E2 -10186.362} C_VEL
LIN {X 0,Y 422.252,Z 448.092,A -85,B 0,C 180,E1 -10186.746,E2 -10186.746} C_VEL
LIN {X 0,Y 423.012,Z 366.587,A -85,B 0,C 180,E1 -10188.146,E2 -10188.146} C_VEL
LIN {X 0,Y 419.462,Z 341.467,A -85,B 0,C 180,E1 -10188.751,E2 -10188.751} C_VEL
LIN {X 0,Y 420.492,Z 323.801,A -85,B 0,C 180,E1 -10192.089,E2 -10192.089} C_VEL
LIN {X 0,Y 421.443,Z 310.443,A -85,B 0,C 180,E1 -10194.638,E2 -10194.638} C_VEL
LIN {X 0,Y 420.442,Z 303.627,A -85,B 0,C 180,E1 -10196.025,E2 -10196.025} C_VEL
LIN {X 0,Y 418.34,Z 293.378,A -85,B 0,C 180,E1 -10198.195,E2 -10198.195} C_VEL
LIN {X 0,Y 418.209,Z 293.388,A -85,B 0,C 180,E1 -10201.395,E2 -10201.395} C_VEL
LIN {X 0,Y 418.262,Z 293.382,A -85,B 0,C 180,E1 -10204.579,E2 -10204.579} C_VEL
LIN {X 0,Y 418.22,Z 293.392,A -85,B 0,C 180,E1 -10207.832,E2 -10207.832} C_VEL
LIN {X 0,Y 418.214,Z 293.387,A -85,B 0,C 180,E1 -10210.947,E2 -10210.947} C_VEL
LIN {X 0,Y 418.203,Z 293.394,A -85,B 0,C 180,E1 -10213.728,E2 -10213.728} C_VEL
LIN {X 0,Y 418.201,Z 293.39,A -85,B 0,C 180,E1 -10216.447,E2 -10216.447} C_VEL
LIN {X 0,Y 418.203,Z 293.39,A -85,B 0,C 180,E1 -10219.132,E2 -10219.132} C_VEL
LIN {X 0,Y 418.232,Z 293.385,A -85,B 0,C 180,E1 -10222.775,E2 -10222.775} C_VEL
LIN {X 0,Y 418.24,Z 293.385,A -85,B 0,C 180,E1 -10226.322,E2 -10226.322} C_VEL
LIN {X 0,Y 418.233,Z 293.389,A -85,B 0,C 180,E1 -10229.727,E2 -10229.727} C_VEL
LIN {X 0,Y 418.202,Z 293.391,A -85,B 0,C 180,E1 -10233.016,E2 -10233.016} C_VEL
LIN {X 0,Y 418.258,Z 293.383,A -85,B 0,C 180,E1 -10236.217,E2 -10236.217} C_VEL
LIN {X 0,Y 418.241,Z 293.39,A -85,B 0,C 180,E1 -10239.337,E2 -10239.337} C_VEL
LIN {X 0,Y 418.27,Z 293.381,A -85,B 0,C 180,E1 -10242.395,E2 -10242.395} C_VEL
LIN {X 0,Y 418.288,Z 293.383,A -85,B 0,C 180,E1 -10245.402,E2 -10245.402} C_VEL
LIN {X 0,Y 418.302,Z 293.377,A -85,B 0,C 180,E1 -10248.369,E2 -10248.369} C_VEL
LIN {X 0,Y 418.367,Z 293.373,A -85,B 0,C 180,E1 -10251.304,E2 -10251.304} C_VEL
LIN {X 0,Y 418.454,Z 293.358,A -85,B 0,C 180,E1 -10254.216,E2 -10254.216} C_VEL
LIN {X 0,Y 418.526,Z 293.35,A -85,B 0,C 180,E1 -10258.075,E2 -10258.075} C_VEL
LIN {X 0,Y 418.462,Z 293.362,A -85,B 0,C 180,E1 -10260.962,E2 -10260.962} C_VEL
LIN {X 0,Y 418.457,Z 293.363,A -85,B 0,C 180,E1 -10262.888,E2 -10262.888} C_VEL
LIN {X 0,Y 418.428,Z 293.364,A -85,B 0,C 180,E1 -10266.605,E2 -10266.605} C_VEL
LIN {X 0,Y 418.325,Z 293.376,A -85,B 0,C 180,E1 -10269.672,E2 -10269.672} C_VEL
LIN {X 0,Y 418.338,Z 293.376,A -85,B 0,C 180,E1 -10273.001,E2 -10273.001} C_VEL
LIN {X 0,Y 418.303,Z 293.381,A -85,B 0,C 180,E1 -10276.735,E2 -10276.735} C_VEL
LIN {X 0,Y 418.262,Z 293.383,A -85,B 0,C 180,E1 -10279.79,E2 -10279.79} C_VEL
LIN {X 0,Y 418.223,Z 293.39,A -85,B 0,C 180,E1 -10282.737,E2 -10282.737} C_VEL
LIN {X 0,Y 418.228,Z 293.387,A -85,B 0,C 180,E1 -10285.907,E2 -10285.907} C_VEL
LIN {X 0,Y 418.253,Z 293.386,A -85,B 0,C 180,E1 -10289.163,E2 -10289.163} C_VEL
LIN {X 0,Y 418.251,Z 293.387,A -85,B 0,C 180,E1 -10292.845,E2 -10292.845} C_VEL
LIN {X 0,Y 418.237,Z 293.389,A -85,B 0,C 180,E1 -10296.239,E2 -10296.239} C_VEL
LIN {X 0,Y 418.236,Z 293.386,A -85,B 0,C 180,E1 -10299.684,E2 -10299.684} C_VEL
LIN {X 0,Y 418.218,Z 293.391,A -85,B 0,C 180,E1 -10302.321,E2 -10302.321} C_VEL
LIN {X 0,Y 418.23,Z 293.387,A -85,B 0,C 180,E1 -10305.11,E2 -10305.11} C_VEL
LIN {X 0,Y 418.235,Z 293.387,A -85,B 0,C 180,E1 -10307.768,E2 -10307.768} C_VEL
LIN {X 0,Y 418.245,Z 293.389,A -85,B 0,C 180,E1 -10310.621,E2 -10310.621} C_VEL
LIN {X 0,Y 418.239,Z 293.388,A -85,B 0,C 180,E1 -10313.977,E2 -10313.977} C_VEL
LIN {X 0,Y 418.254,Z 293.384,A -85,B 0,C 180,E1 -10317.157,E2 -10317.157} C_VEL
LIN {X 0,Y 418.267,Z 293.383,A -85,B 0,C 180,E1 -10320.897,E2 -10320.897} C_VEL
LIN {X 0,Y 418.268,Z 293.385,A -85,B 0,C 180,E1 -10324.097,E2 -10324.097} C_VEL
LIN {X 0,Y 418.237,Z 293.388,A -85,B 0,C 180,E1 -10327.265,E2 -10327.265} C_VEL
LIN {X 0,Y 418.365,Z 293.502,A -85,B 0,C 180,E1 -10330.641,E2 -10330.641} C_VEL
LIN {X 0,Y 419.35,Z 296.95,A -85,B 0,C 180,E1 -10330.9,E2 -10330.9} C_VEL
LIN {X 0,Y 421.172,Z 302.501,A -85,B 0,C 180,E1 -10331.086,E2 -10331.086} C_VEL
LIN {X 0,Y 424.05,Z 323.143,A -85,B 0,C 180,E1 -10331.584,E2 -10331.584} C_VEL
LIN {X 0,Y 422.993,Z 410.753,A -85,B 0,C 180,E1 -10333.098,E2 -10333.098} C_VEL
LIN {X 0,Y 422.693,Z 424.357,A -85,B 0,C 180,E1 -10333.52,E2 -10333.52} C_VEL
LIN {X 0,Y 422.128,Z 436.965,A -85,B 0,C 180,E1 -10334.118,E2 -10334.118} C_VEL
LIN {X 0,Y 421.505,Z 449.092,A -85,B 0,C 180,E1 -10334.9,E2 -10334.9} C_VEL
LIN {X 0,Y 420.949,Z 459.416,A -85,B 0,C 180,E1 -10335.757,E2 -10335.757} C_VEL
LIN {X 0,Y 420.24,Z 469.779,A -85,B 0,C 180,E1 -10336.83,E2 -10336.83} C_VEL
LIN {X 0,Y 419.495,Z 479.509,A -85,B 0,C 180,E1 -10338.076,E2 -10338.076} C_VEL
LIN {X 0,Y 418.922,Z 487.684,A -85,B 0,C 180,E1 -10339.367,E2 -10339.367} C_VEL
LIN {X 0,Y 418.301,Z 495.102,A -85,B 0,C 180,E1 -10340.817,E2 -10340.817} C_VEL
LIN {X 0,Y 418.076,Z 497.841,A -85,B 0,C 180,E1 -10341.443,E2 -10341.443} C_VEL
LIN {X 0,Y 417.21,Z 500.702,A -85,B 0,C 180,E1 -10342.148,E2 -10342.148} C_VEL
LIN {X 0,Y 414.039,Z 504.91,A -85,B 0,C 180,E1 -10343.309,E2 -10343.309} C_VEL
LIN {X 0,Y 410.948,Z 508.416,A -85,B 0,C 180,E1 -10344.528,E2 -10344.528} C_VEL
LIN {X 0,Y 410.221,Z 510.104,A -85,B 0,C 180,E1 -10345.313,E2 -10345.313} C_VEL
LIN {X 0,Y 410.197,Z 512.943,A -85,B 0,C 180,E1 -10347.055,E2 -10347.055} C_VEL
LIN {X 0,Y 409.985,Z 514.554,A -85,B 0,C 180,E1 -10349.019,E2 -10349.019} C_VEL
LIN {X 0,Y 409.976,Z 514.789,A -85,B 0,C 180,E1 -10350.001,E2 -10350.001} C_VEL
LIN {X 0,Y 410.059,Z 514.015,A -85,B 0,C 180,E1 -10351.965,E2 -10351.965} C_VEL
LIN {X 0,Y 410.196,Z 513.049,A -85,B 0,C 180,E1 -10352.947,E2 -10352.947} C_VEL
LIN {X 0,Y 410.225,Z 511.693,A -85,B 0,C 180,E1 -10353.93,E2 -10353.93} C_VEL
LIN {X 0,Y 410.322,Z 508.838,A -85,B 0,C 180,E1 -10355.406,E2 -10355.406} C_VEL
LIN {X 0,Y 410.627,Z 504.796,A -85,B 0,C 180,E1 -10356.932,E2 -10356.932} C_VEL
LIN {X 0,Y 410.936,Z 499.92,A -85,B 0,C 180,E1 -10358.36,E2 -10358.36} C_VEL
LIN {X 0,Y 411.476,Z 493.572,A -85,B 0,C 180,E1 -10359.835,E2 -10359.835} C_VEL
LIN {X 0,Y 412.095,Z 485.674,A -85,B 0,C 180,E1 -10361.311,E2 -10361.311} C_VEL
LIN {X 0,Y 412.77,Z 477.595,A -85,B 0,C 180,E1 -10362.539,E2 -10362.539} C_VEL
LIN {X 0,Y 413.622,Z 467.674,A -85,B 0,C 180,E1 -10363.762,E2 -10363.762} C_VEL
LIN {X 0,Y 414.28,Z 456.532,A -85,B 0,C 180,E1 -10364.869,E2 -10364.869} C_VEL
LIN {X 0,Y 414.939,Z 445.603,A -85,B 0,C 180,E1 -10365.725,E2 -10365.725} C_VEL
LIN {X 0,Y 415.534,Z 433.302,A -85,B 0,C 180,E1 -10366.458,E2 -10366.458} C_VEL
LIN {X 0,Y 416.053,Z 420.504,A -85,B 0,C 180,E1 -10367.005,E2 -10367.005} C_VEL
LIN {X 0,Y 416.32,Z 408.395,A -85,B 0,C 180,E1 -10367.342,E2 -10367.342} C_VEL
LIN {X 0,Y 417.296,Z 322.761,A -85,B 0,C 180,E1 -10368.833,E2 -10368.833} C_VEL
LIN {X 0,Y 414.357,Z 303.172,A -85,B 0,C 180,E1 -10369.328,E2 -10369.328} C_VEL
LIN {X 0,Y 411.837,Z 296.262,A -85,B 0,C 180,E1 -10369.599,E2 -10369.599} C_VEL
LIN {X 0,Y 411.282,Z 294.257,A -85,B 0,C 180,E1 -10369.778,E2 -10369.778} C_VEL
LIN {X 0,Y 411.207,Z 294.261,A -85,B 0,C 180,E1 -10373.148,E2 -10373.148} C_VEL
LIN {X 0,Y 411.242,Z 294.258,A -85,B 0,C 180,E1 -10376.382,E2 -10376.382} C_VEL
LIN {X 0,Y 411.205,Z 294.266,A -85,B 0,C 180,E1 -10379.713,E2 -10379.713} C_VEL
LIN {X 0,Y 411.211,Z 294.262,A -85,B 0,C 180,E1 -10383.156,E2 -10383.156} C_VEL
LIN {X 0,Y 411.197,Z 294.262,A -85,B 0,C 180,E1 -10386.553,E2 -10386.553} C_VEL
LIN {X 0,Y 411.22,Z 294.262,A -85,B 0,C 180,E1 -10389.729,E2 -10389.729} C_VEL
LIN {X 0,Y 411.183,Z 294.268,A -85,B 0,C 180,E1 -10393.133,E2 -10393.133} C_VEL
LIN {X 0,Y 411.174,Z 294.266,A -85,B 0,C 180,E1 -10395.881,E2 -10395.881} C_VEL
LIN {X 0,Y 411.168,Z 294.267,A -85,B 0,C 180,E1 -10398.772,E2 -10398.772} C_VEL
LIN {X 0,Y 411.209,Z 294.26,A -85,B 0,C 180,E1 -10401.832,E2 -10401.832} C_VEL
LIN {X 0,Y 411.216,Z 294.264,A -85,B 0,C 180,E1 -10405.122,E2 -10405.122} C_VEL
LIN {X 0,Y 411.171,Z 294.264,A -85,B 0,C 180,E1 -10408.003,E2 -10408.003} C_VEL
LIN {X 0,Y 411.222,Z 294.259,A -85,B 0,C 180,E1 -10411.41,E2 -10411.41} C_VEL
LIN {X 0,Y 411.239,Z 294.256,A -85,B 0,C 180,E1 -10413.619,E2 -10413.619} C_VEL
LIN {X 0,Y 411.207,Z 294.265,A -85,B 0,C 180,E1 -10416.853,E2 -10416.853} C_VEL
LIN {X 0,Y 411.253,Z 294.313,A -85,B 0,C 180,E1 -10418.641,E2 -10418.641} C_VEL
LIN {X 0,Y 412.654,Z 302.978,A -85,B 0,C 180,E1 -10420.861,E2 -10420.861} C_VEL
LIN {X 0,Y 412.642,Z 304.21,A -85,B 0,C 180,E1 -10421.162,E2 -10421.162} C_VEL
LIN {X 0,Y 416.282,Z 323.862,A -85,B 0,C 180,E1 -10421.737,E2 -10421.737} C_VEL
LIN {X 0,Y 414.622,Z 412.565,A -85,B 0,C 180,E1 -10423.632,E2 -10423.632} C_VEL
LIN {X 0,Y 414.314,Z 426.161,A -85,B 0,C 180,E1 -10424.126,E2 -10424.126} C_VEL
LIN {X 0,Y 413.75,Z 438.051,A -85,B 0,C 180,E1 -10424.735,E2 -10424.735} C_VEL
LIN {X 0,Y 413.323,Z 449.911,A -85,B 0,C 180,E1 -10425.545,E2 -10425.545} C_VEL
LIN {X 0,Y 412.736,Z 461.906,A -85,B 0,C 180,E1 -10426.585,E2 -10426.585} C_VEL
LIN {X 0,Y 412.173,Z 472.093,A -85,B 0,C 180,E1 -10427.694,E2 -10427.694} C_VEL
LIN {X 0,Y 411.607,Z 481.339,A -85,B 0,C 180,E1 -10428.925,E2 -10428.925} C_VEL
LIN {X 0,Y 411.118,Z 490.368,A -85,B 0,C 180,E1 -10430.405,E2 -10430.405} C_VEL
LIN {X 0,Y 410.697,Z 497.545,A -85,B 0,C 180,E1 -10431.884,E2 -10431.884} C_VEL
LIN {X 0,Y 410.415,Z 504.123,A -85,B 0,C 180,E1 -10433.607,E2 -10433.607} C_VEL
LIN {X 0,Y 410.211,Z 508.428,A -85,B 0,C 180,E1 -10435.086,E2 -10435.086} C_VEL
LIN {X 0,Y 410.172,Z 510.647,A -85,B 0,C 180,E1 -10436.07,E2 -10436.07} C_VEL
LIN {X 0,Y 410.171,Z 512.409,A -85,B 0,C 180,E1 -10437.053,E2 -10437.053} C_VEL
LIN {X 0,Y 410.059,Z 513.756,A -85,B 0,C 180,E1 -10438.036,E2 -10438.036} C_VEL
LIN {X 0,Y 409.987,Z 514.646,A -85,B 0,C 180,E1 -10439.018,E2 -10439.018} C_VEL
LIN {X 0,Y 409.979,Z 515.095,A -85,B 0,C 180,E1 -10440,E2 -10440} C_VEL
LIN {X 0,Y 410.011,Z 515.135,A -85,B 0,C 180,E1 -10440.982,E2 -10440.982} C_VEL
LIN {X 0,Y 410.087,Z 514.759,A -85,B 0,C 180,E1 -10441.964,E2 -10441.964} C_VEL
LIN {X 0,Y 410.211,Z 513.914,A -85,B 0,C 180,E1 -10442.946,E2 -10442.946} C_VEL
LIN {X 0,Y 410.354,Z 512.652,A -85,B 0,C 180,E1 -10443.928,E2 -10443.928} C_VEL
LIN {X 0,Y 410.34,Z 509.944,A -85,B 0,C 180,E1 -10445.405,E2 -10445.405} C_VEL
LIN {X 0,Y 410.762,Z 506.137,A -85,B 0,C 180,E1 -10446.879,E2 -10446.879} C_VEL
LIN {X 0,Y 411.071,Z 501.186,A -85,B 0,C 180,E1 -10448.356,E2 -10448.356} C_VEL
LIN {X 0,Y 411.65,Z 494.91,A -85,B 0,C 180,E1 -10449.83,E2 -10449.83} C_VEL
LIN {X 0,Y 412.247,Z 487.021,A -85,B 0,C 180,E1 -10451.306,E2 -10451.306} C_VEL
LIN {X 0,Y 412.81,Z 478.976,A -85,B 0,C 180,E1 -10452.537,E2 -10452.537} C_VEL
LIN {X 0,Y 413.611,Z 469.172,A -85,B 0,C 180,E1 -10453.762,E2 -10453.762} C_VEL
LIN {X 0,Y 414.441,Z 458.348,A -85,B 0,C 180,E1 -10454.849,E2 -10454.849} C_VEL
LIN {X 0,Y 415.225,Z 445.907,A -85,B 0,C 180,E1 -10455.839,E2 -10455.839} C_VEL
LIN {X 0,Y 415.888,Z 433.954,A -85,B 0,C 180,E1 -10456.569,E2 -10456.569} C_VEL
LIN {X 0,Y 416.416,Z 421.073,A -85,B 0,C 180,E1 -10457.147,E2 -10457.147} C_VEL
LIN {X 0,Y 416.819,Z 407.961,A -85,B 0,C 180,E1 -10457.541,E2 -10457.541} C_VEL
LIN {X 0,Y 419.393,Z 326.448,A -85,B 0,C 180,E1 -10459.481,E2 -10459.481} C_VEL
LIN {X 0,Y 418.155,Z 320.177,A -85,B 0,C 180,E1 -10459.744,E2 -10459.744} C_VEL
LIN {X 0,Y 415.56,Z 311.801,A -85,B 0,C 180,E1 -10460.178,E2 -10460.178} C_VEL
LIN {X 0,Y 414.239,Z 308.416,A -85,B 0,C 180,E1 -10460.396,E2 -10460.396} C_VEL
LIN {X 0,Y 412.608,Z 300.123,A -85,B 0,C 180,E1 -10463.103,E2 -10463.103} C_VEL
LIN {X 0,Y 411.183,Z 294.27,A -85,B 0,C 180,E1 -10465.212,E2 -10465.212} C_VEL
LIN {X 0,Y 411.171,Z 294.27,A -85,B 0,C 180,E1 -10468.594,E2 -10468.594} C_VEL
LIN {X 0,Y 411.157,Z 294.27,A -85,B 0,C 180,E1 -10471.998,E2 -10471.998} C_VEL
LIN {X 0,Y 411.203,Z 294.267,A -85,B 0,C 180,E1 -10474.876,E2 -10474.876} C_VEL
LIN {X 0,Y 411.192,Z 294.266,A -85,B 0,C 180,E1 -10478.165,E2 -10478.165} C_VEL
LIN {X 0,Y 411.163,Z 294.268,A -85,B 0,C 180,E1 -10481.807,E2 -10481.807} C_VEL
LIN {X 0,Y 411.176,Z 294.266,A -85,B 0,C 180,E1 -10485.509,E2 -10485.509} C_VEL
LIN {X 0,Y 411.15,Z 294.271,A -85,B 0,C 180,E1 -10488.774,E2 -10488.774} C_VEL
LIN {X 0,Y 411.188,Z 294.268,A -85,B 0,C 180,E1 -10492.025,E2 -10492.025} C_VEL
LIN {X 0,Y 411.209,Z 294.265,A -85,B 0,C 180,E1 -10495.666,E2 -10495.666} C_VEL
LIN {X 0,Y 411.207,Z 294.306,A -85,B 0,C 180,E1 -10499.044,E2 -10499.044} C_VEL
LIN {X 0,Y 413.862,Z 304.382,A -85,B 0,C 180,E1 -10502.011,E2 -10502.011} C_VEL
LIN {X 0,Y 415.671,Z 313.856,A -85,B 0,C 180,E1 -10504.459,E2 -10504.459} C_VEL
LIN {X 0,Y 415.218,Z 319.776,A -85,B 0,C 180,E1 -10505.766,E2 -10505.766} C_VEL
LIN {X 0,Y 413.907,Z 333.167,A -85,B 0,C 180,E1 -10508.588,E2 -10508.588} C_VEL
LIN {X 0,Y 413.469,Z 337.927,A -85,B 0,C 180,E1 -10509.565,E2 -10509.565} C_VEL
LIN {X 0,Y 416.626,Z 353.923,A -85,B 0,C 180,E1 -10510.247,E2 -10510.247} C_VEL
LIN {X 0,Y 418.458,Z 368.928,A -85,B 0,C 180,E1 -10510.776,E2 -10510.776} C_VEL
LIN {X 0,Y 416.106,Z 450.419,A -85,B 0,C 180,E1 -10512.712,E2 -10512.712} C_VEL
LIN {X 0,Y 415.395,Z 463.809,A -85,B 0,C 180,E1 -10513.22,E2 -10513.22} C_VEL
LIN {X 0,Y 414.62,Z 476.167,A -85,B 0,C 180,E1 -10513.884,E2 -10513.884} C_VEL
LIN {X 0,Y 413.802,Z 488.316,A -85,B 0,C 180,E1 -10514.736,E2 -10514.736} C_VEL
LIN {X 0,Y 412.994,Z 499.355,A -85,B 0,C 180,E1 -10515.714,E2 -10515.714} C_VEL
LIN {X 0,Y 412.107,Z 510.653,A -85,B 0,C 180,E1 -10516.966,E2 -10516.966} C_VEL
LIN {X 0,Y 411.546,Z 519.53,A -85,B 0,C 180,E1 -10518.174,E2 -10518.174} C_VEL
LIN {X 0,Y 410.843,Z 528.391,A -85,B 0,C 180,E1 -10519.652,E2 -10519.652} C_VEL
LIN {X 0,Y 410.447,Z 535.536,A -85,B 0,C 180,E1 -10521.134,E2 -10521.134} C_VEL
LIN {X 0,Y 410.176,Z 541.262,A -85,B 0,C 180,E1 -10522.616,E2 -10522.616} C_VEL
LIN {X 0,Y 410.016,Z 545.744,A -85,B 0,C 180,E1 -10524.096,E2 -10524.096} C_VEL
LIN {X 0,Y 410.027,Z 548.123,A -85,B 0,C 180,E1 -10525.083,E2 -10525.083} C_VEL
LIN {X 0,Y 409.943,Z 549.982,A -85,B 0,C 180,E1 -10526.067,E2 -10526.067} C_VEL
LIN {X 0,Y 409.969,Z 551.413,A -85,B 0,C 180,E1 -10527.051,E2 -10527.051} C_VEL
LIN {X 0,Y 410.018,Z 552.421,A -85,B 0,C 180,E1 -10528.034,E2 -10528.034} C_VEL
LIN {X 0,Y 409.979,Z 552.951,A -85,B 0,C 180,E1 -10529.017,E2 -10529.017} C_VEL
LIN {X 0,Y 409.984,Z 553.05,A -85,B 0,C 180,E1 -10529.999,E2 -10529.999} C_VEL
LIN {X 0,Y 409.979,Z 552.73,A -85,B 0,C 180,E1 -10530.981,E2 -10530.981} C_VEL
LIN {X 0,Y 410.022,Z 551.977,A -85,B 0,C 180,E1 -10531.964,E2 -10531.964} C_VEL
LIN {X 0,Y 410.024,Z 550.741,A -85,B 0,C 180,E1 -10532.947,E2 -10532.947} C_VEL
LIN {X 0,Y 410.007,Z 548.058,A -85,B 0,C 180,E1 -10534.423,E2 -10534.423} C_VEL
LIN {X 0,Y 410.055,Z 544.28,A -85,B 0,C 180,E1 -10535.901,E2 -10535.901} C_VEL
LIN {X 0,Y 410.259,Z 537.668,A -85,B 0,C 180,E1 -10537.876,E2 -10537.876} C_VEL
LIN {X 0,Y 410.522,Z 531.536,A -85,B 0,C 180,E1 -10539.359,E2 -10539.359} C_VEL
LIN {X 0,Y 410.922,Z 523.898,A -85,B 0,C 180,E1 -10540.843,E2 -10540.843} C_VEL
LIN {X 0,Y 411.561,Z 516.063,A -85,B 0,C 180,E1 -10542.074,E2 -10542.074} C_VEL
LIN {X 0,Y 412.17,Z 507.043,A -85,B 0,C 180,E1 -10543.24,E2 -10543.24} C_VEL
LIN {X 0,Y 412.937,Z 495.81,A -85,B 0,C 180,E1 -10544.412,E2 -10544.412} C_VEL
LIN {X 0,Y 413.586,Z 485.466,A -85,B 0,C 180,E1 -10545.27,E2 -10545.27} C_VEL
LIN {X 0,Y 414.356,Z 473.02,A -85,B 0,C 180,E1 -10546.061,E2 -10546.061} C_VEL
LIN {X 0,Y 414.956,Z 460.638,A -85,B 0,C 180,E1 -10546.638,E2 -10546.638} C_VEL
LIN {X 0,Y 415.471,Z 447.85,A -85,B 0,C 180,E1 -10547.028,E2 -10547.028} C_VEL
LIN {X 0,Y 416.208,Z 366.943,A -85,B 0,C 180,E1 -10548.443,E2 -10548.443} C_VEL
LIN {X 0,Y 412.501,Z 340.672,A -85,B 0,C 180,E1 -10549.112,E2 -10549.112} C_VEL
LIN {X 0,Y 413.586,Z 323.173,A -85,B 0,C 180,E1 -10552.477,E2 -10552.477} C_VEL
LIN {X 0,Y 414.47,Z 311.175,A -85,B 0,C 180,E1 -10554.813,E2 -10554.813} C_VEL
LIN {X 0,Y 413.08,Z 302.986,A -85,B 0,C 180,E1 -10556.525,E2 -10556.525} C_VEL
LIN {X 0,Y 411.297,Z 294.255,A -85,B 0,C 180,E1 -10558.443,E2 -10558.443} C_VEL
LIN {X 0,Y 411.163,Z 294.271,A -85,B 0,C 180,E1 -10561.996,E2 -10561.996} C_VEL
LIN {X 0,Y 411.207,Z 294.26,A -85,B 0,C 180,E1 -10564.877,E2 -10564.877} C_VEL
LIN {X 0,Y 411.194,Z 294.266,A -85,B 0,C 180,E1 -10568.166,E2 -10568.166} C_VEL
LIN {X 0,Y 411.155,Z 294.267,A -85,B 0,C 180,E1 -10571.227,E2 -10571.227} C_VEL
LIN {X 0,Y 411.17,Z 294.266,A -85,B 0,C 180,E1 -10574.489,E2 -10574.489} C_VEL
LIN {X 0,Y 411.163,Z 294.268,A -85,B 0,C 180,E1 -10578.193,E2 -10578.193} C_VEL
LIN {X 0,Y 411.188,Z 294.267,A -85,B 0,C 180,E1 -10581.832,E2 -10581.832} C_VEL
LIN {X 0,Y 411.203,Z 294.262,A -85,B 0,C 180,E1 -10585.121,E2 -10585.121} C_VEL
LIN {X 0,Y 411.157,Z 294.269,A -85,B 0,C 180,E1 -10588.002,E2 -10588.002} C_VEL
LIN {X 0,Y 411.168,Z 294.27,A -85,B 0,C 180,E1 -10591.406,E2 -10591.406} C_VEL
LIN {X 0,Y 411.204,Z 294.262,A -85,B 0,C 180,E1 -10594.933,E2 -10594.933} C_VEL
LIN {X 0,Y 411.195,Z 294.265,A -85,B 0,C 180,E1 -10597.913,E2 -10597.913} C_VEL
LIN {X 0,Y 411.21,Z 294.263,A -85,B 0,C 180,E1 -10601.051,E2 -10601.051} C_VEL
LIN {X 0,Y 411.243,Z 294.257,A -85,B 0,C 180,E1 -10604.131,E2 -10604.131} C_VEL
LIN {X 0,Y 411.294,Z 294.255,A -85,B 0,C 180,E1 -10607.165,E2 -10607.165} C_VEL
LIN {X 0,Y 411.279,Z 294.252,A -85,B 0,C 180,E1 -10610.161,E2 -10610.161} C_VEL
LIN {X 0,Y 411.376,Z 294.245,A -85,B 0,C 180,E1 -10613.132,E2 -10613.132} C_VEL
LIN {X 0,Y 411.275,Z 294.257,A -85,B 0,C 180,E1 -10615.099,E2 -10615.099} C_VEL
LIN {X 0,Y 411.495,Z 294.225,A -85,B 0,C 180,E1 -10618.043,E2 -10618.043} C_VEL
LIN {X 0,Y 411.491,Z 294.226,A -85,B 0,C 180,E1 -10621.958,E2 -10621.958} C_VEL
LIN {X 0,Y 411.376,Z 294.242,A -85,B 0,C 180,E1 -10626.606,E2 -10626.606} C_VEL
LIN {X 0,Y 411.278,Z 294.253,A -85,B 0,C 180,E1 -10629.839,E2 -10629.839} C_VEL
LIN {X 0,Y 411.297,Z 294.253,A -85,B 0,C 180,E1 -10633.104,E2 -10633.104} C_VEL
LIN {X 0,Y 411.249,Z 294.259,A -85,B 0,C 180,E1 -10636.889,E2 -10636.889} C_VEL
LIN {X 0,Y 411.222,Z 294.259,A -85,B 0,C 180,E1 -10639.987,E2 -10639.987} C_VEL
LIN {X 0,Y 411.187,Z 294.267,A -85,B 0,C 180,E1 -10643.149,E2 -10643.149} C_VEL
LIN {X 0,Y 411.195,Z 294.266,A -85,B 0,C 180,E1 -10646.384,E2 -10646.384} C_VEL
LIN {X 0,Y 411.19,Z 294.263,A -85,B 0,C 180,E1 -10649.714,E2 -10649.714} C_VEL
LIN {X 0,Y 411.2,Z 294.264,A -85,B 0,C 180,E1 -10653.157,E2 -10653.157} C_VEL
LIN {X 0,Y 411.185,Z 294.267,A -85,B 0,C 180,E1 -10656.553,E2 -10656.553} C_VEL
LIN {X 0,Y 411.201,Z 294.262,A -85,B 0,C 180,E1 -10659.728,E2 -10659.728} C_VEL
LIN {X 0,Y 411.165,Z 294.267,A -85,B 0,C 180,E1 -10663.135,E2 -10663.135} C_VEL
LIN {X 0,Y 411.163,Z 294.268,A -85,B 0,C 180,E1 -10665.882,E2 -10665.882} C_VEL
LIN {X 0,Y 411.159,Z 294.27,A -85,B 0,C 180,E1 -10668.773,E2 -10668.773} C_VEL
LIN {X 0,Y 411.189,Z 294.267,A -85,B 0,C 180,E1 -10672.027,E2 -10672.027} C_VEL
LIN {X 0,Y 411.201,Z 294.263,A -85,B 0,C 180,E1 -10675.667,E2 -10675.667} C_VEL
LIN {X 0,Y 411.187,Z 294.264,A -85,B 0,C 180,E1 -10679.154,E2 -10679.154} C_VEL
LIN {X 0,Y 411.257,Z 294.258,A -85,B 0,C 180,E1 -10682.524,E2 -10682.524} C_VEL
LIN {X 0,Y 411.226,Z 294.262,A -85,B 0,C 180,E1 -10685.786,E2 -10685.786} C_VEL
LIN {X 0,Y 411.202,Z 294.266,A -85,B 0,C 180,E1 -10688.967,E2 -10688.967} C_VEL
LIN {X 0,Y 411.288,Z 294.393,A -85,B 0,C 180,E1 -10690.346,E2 -10690.346} C_VEL
LIN {X 0,Y 412.28,Z 297.571,A -85,B 0,C 180,E1 -10690.566,E2 -10690.566} C_VEL
LIN {X 0,Y 414.677,Z 304.546,A -85,B 0,C 180,E1 -10690.811,E2 -10690.811} C_VEL
LIN {X 0,Y 417.324,Z 323.368,A -85,B 0,C 180,E1 -10691.276,E2 -10691.276} C_VEL
LIN {X 0,Y 416.203,Z 412.298,A -85,B 0,C 180,E1 -10692.845,E2 -10692.845} C_VEL
LIN {X 0,Y 415.876,Z 425.37,A -85,B 0,C 180,E1 -10693.274,E2 -10693.274} C_VEL
LIN {X 0,Y 415.255,Z 438.327,A -85,B 0,C 180,E1 -10693.912,E2 -10693.912} C_VEL
LIN {X 0,Y 414.584,Z 450.998,A -85,B 0,C 180,E1 -10694.768,E2 -10694.768} C_VEL
LIN {X 0,Y 413.993,Z 461.772,A -85,B 0,C 180,E1 -10695.718,E2 -10695.718} C_VEL
LIN {X 0,Y 413.177,Z 472.156,A -85,B 0,C 180,E1 -10696.851,E2 -10696.851} C_VEL
LIN {X 0,Y 412.52,Z 480.399,A -85,B 0,C 180,E1 -10697.955,E2 -10697.955} C_VEL
LIN {X 0,Y 411.824,Z 489.329,A -85,B 0,C 180,E1 -10699.43,E2 -10699.43} C_VEL
LIN {X 0,Y 411.214,Z 496.503,A -85,B 0,C 180,E1 -10700.905,E2 -10700.905} C_VEL
LIN {X 0,Y 410.743,Z 503.087,A -85,B 0,C 180,E1 -10702.629,E2 -10702.629} C_VEL
LIN {X 0,Y 410.482,Z 507.403,A -85,B 0,C 180,E1 -10704.105,E2 -10704.105} C_VEL
LIN {X 0,Y 410.221,Z 510.104,A -85,B 0,C 180,E1 -10705.313,E2 -10705.313} C_VEL
LIN {X 0,Y 409.516,Z 511.637,A -85,B 0,C 180,E1 -10706.109,E2 -10706.109} C_VEL
LIN {X 0,Y 406.545,Z 513.528,A -85,B 0,C 180,E1 -10707.411,E2 -10707.411} C_VEL
LIN {X 0,Y 404.045,Z 514.566,A -85,B 0,C 180,E1 -10708.474,E2 -10708.474} C_VEL
LIN {X 0,Y 402.91,Z 515.018,A -85,B 0,C 180,E1 -10709.443,E2 -10709.443} C_VEL
LIN {X 0,Y 402.889,Z 515.007,A -85,B 0,C 180,E1 -10709.583,E2 -10709.583} C_VEL
LIN {X 0,Y 402.911,Z 514.915,A -85,B 0,C 180,E1 -10711,E2 -10711} C_VEL
LIN {X 0,Y 403.133,Z 513.364,A -85,B 0,C 180,E1 -10712.999,E2 -10712.999} C_VEL
LIN {X 0,Y 403.135,Z 512.009,A -85,B 0,C 180,E1 -10714,E2 -10714} C_VEL
LIN {X 0,Y 403.28,Z 509.152,A -85,B 0,C 180,E1 -10715.501,E2 -10715.501} C_VEL
LIN {X 0,Y 403.567,Z 505.264,A -85,B 0,C 180,E1 -10717.003,E2 -10717.003} C_VEL
LIN {X 0,Y 403.907,Z 500.233,A -85,B 0,C 180,E1 -10718.506,E2 -10718.506} C_VEL
LIN {X 0,Y 404.494,Z 493.883,A -85,B 0,C 180,E1 -10720.007,E2 -10720.007} C_VEL
LIN {X 0,Y 405.144,Z 485.983,A -85,B 0,C 180,E1 -10721.508,E2 -10721.508} C_VEL
LIN {X 0,Y 405.858,Z 477.901,A -85,B 0,C 180,E1 -10722.756,E2 -10722.756} C_VEL
LIN {X 0,Y 406.749,Z 467.976,A -85,B 0,C 180,E1 -10724,E2 -10724} C_VEL
LIN {X 0,Y 407.433,Z 456.829,A -85,B 0,C 180,E1 -10725.124,E2 -10725.124} C_VEL
LIN {X 0,Y 408.117,Z 445.893,A -85,B 0,C 180,E1 -10725.994,E2 -10725.994} C_VEL
LIN {X 0,Y 408.742,Z 433.578,A -85,B 0,C 180,E1 -10726.739,E2 -10726.739} C_VEL
LIN {X 0,Y 409.285,Z 420.759,A -85,B 0,C 180,E1 -10727.295,E2 -10727.295} C_VEL
LIN {X 0,Y 409.551,Z 408.592,A -85,B 0,C 180,E1 -10727.638,E2 -10727.638} C_VEL
LIN {X 0,Y 410.599,Z 323.617,A -85,B 0,C 180,E1 -10729.14,E2 -10729.14} C_VEL
LIN {X 0,Y 407.752,Z 304.821,A -85,B 0,C 180,E1 -10729.626,E2 -10729.626} C_VEL
LIN {X 0,Y 404.498,Z 296.396,A -85,B 0,C 180,E1 -10729.973,E2 -10729.973} C_VEL
LIN {X 0,Y 404.22,Z 295.135,A -85,B 0,C 180,E1 -10730.085,E2 -10730.085} C_VEL
LIN {X 0,Y 404.173,Z 295.14,A -85,B 0,C 180,E1 -10733.575,E2 -10733.575} C_VEL
LIN {X 0,Y 404.188,Z 295.141,A -85,B 0,C 180,E1 -10735.767,E2 -10735.767} C_VEL
LIN {X 0,Y 404.2,Z 295.137,A -85,B 0,C 180,E1 -10738,E2 -10738} C_VEL
LIN {X 0,Y 404.144,Z 295.146,A -85,B 0,C 180,E1 -10741.558,E2 -10741.558} C_VEL
LIN {X 0,Y 404.188,Z 295.136,A -85,B 0,C 180,E1 -10745.017,E2 -10745.017} C_VEL
LIN {X 0,Y 404.161,Z 295.139,A -85,B 0,C 180,E1 -10748.757,E2 -10748.757} C_VEL
LIN {X 0,Y 404.129,Z 295.146,A -85,B 0,C 180,E1 -10751.6,E2 -10751.6} C_VEL
LIN {X 0,Y 404.154,Z 295.139,A -85,B 0,C 180,E1 -10754.523,E2 -10754.523} C_VEL
LIN {X 0,Y 404.141,Z 295.146,A -85,B 0,C 180,E1 -10757.296,E2 -10757.296} C_VEL
LIN {X 0,Y 404.174,Z 295.137,A -85,B 0,C 180,E1 -10759.956,E2 -10759.956} C_VEL
LIN {X 0,Y 404.142,Z 295.146,A -85,B 0,C 180,E1 -10763.125,E2 -10763.125} C_VEL
LIN {X 0,Y 404.15,Z 295.139,A -85,B 0,C 180,E1 -10766.188,E2 -10766.188} C_VEL
LIN {X 0,Y 404.151,Z 295.139,A -85,B 0,C 180,E1 -10769.715,E2 -10769.715} C_VEL
LIN {X 0,Y 404.198,Z 295.136,A -85,B 0,C 180,E1 -10773.123,E2 -10773.123} C_VEL
LIN {X 0,Y 404.178,Z 295.137,A -85,B 0,C 180,E1 -10775.334,E2 -10775.334} C_VEL
LIN {X 0,Y 404.218,Z 295.28,A -85,B 0,C 180,E1 -10778.518,E2 -10778.518} C_VEL
LIN {X 0,Y 405.559,Z 302.945,A -85,B 0,C 180,E1 -10780.513,E2 -10780.513} C_VEL
LIN {X 0,Y 405.683,Z 304.66,A -85,B 0,C 180,E1 -10780.911,E2 -10780.911} C_VEL
LIN {X 0,Y 409.391,Z 325.153,A -85,B 0,C 180,E1 -10781.519,E2 -10781.519} C_VEL
LIN {X 0,Y 407.669,Z 412.704,A -85,B 0,C 180,E1 -10783.442,E2 -10783.442} C_VEL
LIN {X 0,Y 407.299,Z 427.025,A -85,B 0,C 180,E1 -10783.973,E2 -10783.973} C_VEL
LIN {X 0,Y 406.754,Z 438.732,A -85,B 0,C 180,E1 -10784.594,E2 -10784.594} C_VEL
LIN {X 0,Y 406.25,Z 451.593,A -85,B 0,C 180,E1 -10785.503,E2 -10785.503} C_VEL
LIN {X 0,Y 405.71,Z 462.461,A -85,B 0,C 180,E1 -10786.476,E2 -10786.476} C_VEL
LIN {X 0,Y 405.124,Z 472.606,A -85,B 0,C 180,E1 -10787.603,E2 -10787.603} C_VEL
LIN {X 0,Y 404.487,Z 482.677,A -85,B 0,C 180,E1 -10788.981,E2 -10788.981} C_VEL
LIN {X 0,Y 404.074,Z 490.162,A -85,B 0,C 180,E1 -10790.236,E2 -10790.236} C_VEL
LIN {X 0,Y 403.664,Z 497.477,A -85,B 0,C 180,E1 -10791.742,E2 -10791.742} C_VEL
LIN {X 0,Y 403.4,Z 503.305,A -85,B 0,C 180,E1 -10793.245,E2 -10793.245} C_VEL
LIN {X 0,Y 403.151,Z 508.532,A -85,B 0,C 180,E1 -10794.999,E2 -10794.999} C_VEL
LIN {X 0,Y 403.079,Z 510.823,A -85,B 0,C 180,E1 -10796.001,E2 -10796.001} C_VEL
LIN {X 0,Y 403.089,Z 512.62,A -85,B 0,C 180,E1 -10797.002,E2 -10797.002} C_VEL
LIN {X 0,Y 402.991,Z 513.999,A -85,B 0,C 180,E1 -10798.001,E2 -10798.001} C_VEL
LIN {X 0,Y 402.912,Z 514.949,A -85,B 0,C 180,E1 -10799,E2 -10799} C_VEL
LIN {X 0,Y 402.901,Z 515.431,A -85,B 0,C 180,E1 -10800,E2 -10800} C_VEL
LIN {X 0,Y 402.935,Z 515.503,A -85,B 0,C 180,E1 -10800.999,E2 -10800.999} C_VEL
LIN {X 0,Y 403.018,Z 515.164,A -85,B 0,C 180,E1 -10801.999,E2 -10801.999} C_VEL
LIN {X 0,Y 403.153,Z 514.363,A -85,B 0,C 180,E1 -10802.998,E2 -10802.998} C_VEL
LIN {X 0,Y 403.298,Z 513.128,A -85,B 0,C 180,E1 -10803.997,E2 -10803.997} C_VEL
LIN {X 0,Y 403.296,Z 510.478,A -85,B 0,C 180,E1 -10805.5,E2 -10805.5} C_VEL
LIN {X 0,Y 403.783,Z 506.157,A -85,B 0,C 180,E1 -10807.199,E2 -10807.199} C_VEL
LIN {X 0,Y 404.091,Z 501.829,A -85,B 0,C 180,E1 -10808.501,E2 -10808.501} C_VEL
LIN {X 0,Y 404.707,Z 495.622,A -85,B 0,C 180,E1 -10810,E2 -10810} C_VEL
LIN {X 0,Y 405.341,Z 487.85,A -85,B 0,C 180,E1 -10811.501,E2 -10811.501} C_VEL
LIN {X 0,Y 405.949,Z 479.888,A -85,B 0,C 180,E1 -10812.752,E2 -10812.752} C_VEL
LIN {X 0,Y 406.793,Z 470.209,A -85,B 0,C 180,E1 -10813.997,E2 -10813.997} C_VEL
LIN {X 0,Y 407.714,Z 459.23,A -85,B 0,C 180,E1 -10815.135,E2 -10815.135} C_VEL
LIN {X 0,Y 408.522,Z 447.387,A -85,B 0,C 180,E1 -10816.105,E2 -10816.105} C_VEL
LIN {X 0,Y 409.275,Z 434.755,A -85,B 0,C 180,E1 -10816.909,E2 -10816.909} C_VEL
LIN {X 0,Y 409.83,Z 422.132,A -85,B 0,C 180,E1 -10817.496,E2 -10817.496} C_VEL
LIN {X 0,Y 410.314,Z 408.33,A -85,B 0,C 180,E1 -10817.925,E2 -10817.925} C_VEL
LIN {X 0,Y 413.05,Z 328.393,A -85,B 0,C 180,E1 -10819.895,E2 -10819.895} C_VEL
LIN {X 0,Y 412.783,Z 325.466,A -85,B 0,C 180,E1 -10819.999,E2 -10819.999} C_VEL
LIN {X 0,Y 410.303,Z 316.405,A -85,B 0,C 180,E1 -10820.461,E2 -10820.461} C_VEL
LIN {X 0,Y 407.29,Z 309.012,A -85,B 0,C 180,E1 -10820.953,E2 -10820.953} C_VEL
LIN {X 0,Y 405.358,Z 300.054,A -85,B 0,C 180,E1 -10824.044,E2 -10824.044} C_VEL
LIN {X 0,Y 404.111,Z 295.151,A -85,B 0,C 180,E1 -10825.979,E2 -10825.979} C_VEL
LIN {X 0,Y 404.154,Z 295.143,A -85,B 0,C 180,E1 -10829.601,E2 -10829.601} C_VEL
LIN {X 0,Y 404.17,Z 295.142,A -85,B 0,C 180,E1 -10833.418,E2 -10833.418} C_VEL
LIN {X 0,Y 404.136,Z 295.145,A -85,B 0,C 180,E1 -10836.247,E2 -10836.247} C_VEL
LIN {X 0,Y 404.135,Z 295.145,A -85,B 0,C 180,E1 -10838.759,E2 -10838.759} C_VEL
LIN {X 0,Y 404.109,Z 295.147,A -85,B 0,C 180,E1 -10841.596,E2 -10841.596} C_VEL
LIN {X 0,Y 404.146,Z 295.144,A -85,B 0,C 180,E1 -10844.521,E2 -10844.521} C_VEL
LIN {X 0,Y 404.123,Z 295.145,A -85,B 0,C 180,E1 -10847.293,E2 -10847.293} C_VEL
LIN {X 0,Y 404.136,Z 295.144,A -85,B 0,C 180,E1 -10849.95,E2 -10849.95} C_VEL
LIN {X 0,Y 404.137,Z 295.145,A -85,B 0,C 180,E1 -10853.125,E2 -10853.125} C_VEL
LIN {X 0,Y 404.149,Z 295.147,A -85,B 0,C 180,E1 -10856.187,E2 -10856.187} C_VEL
LIN {X 0,Y 404.142,Z 295.166,A -85,B 0,C 180,E1 -10858.319,E2 -10858.319} C_VEL
LIN {X 0,Y 406.478,Z 303.796,A -85,B 0,C 180,E1 -10861.044,E2 -10861.044} C_VEL
LIN {X 0,Y 408.385,Z 312.616,A -85,B 0,C 180,E1 -10863.493,E2 -10863.493} C_VEL
LIN {X 0,Y 408.987,Z 316.84,A -85,B 0,C 180,E1 -10864.557,E2 -10864.557} C_VEL
LIN {X 0,Y 407.285,Z 332.363,A -85,B 0,C 180,E1 -10867.955,E2 -10867.955} C_VEL
LIN {X 0,Y 406.775,Z 337.493,A -85,B 0,C 180,E1 -10869.036,E2 -10869.036} C_VEL
LIN {X 0,Y 410.135,Z 354.165,A -85,B 0,C 180,E1 -10869.784,E2 -10869.784} C_VEL
LIN {X 0,Y 412.029,Z 369.194,A -85,B 0,C 180,E1 -10870.345,E2 -10870.345} C_VEL
LIN {X 0,Y 409.529,Z 449.809,A -85,B 0,C 180,E1 -10872.329,E2 -10872.329} C_VEL
LIN {X 0,Y 408.858,Z 462.459,A -85,B 0,C 180,E1 -10872.815,E2 -10872.815} C_VEL
LIN {X 0,Y 407.998,Z 475.037,A -85,B 0,C 180,E1 -10873.487,E2 -10873.487} C_VEL
LIN {X 0,Y 407.118,Z 487.275,A -85,B 0,C 180,E1 -10874.351,E2 -10874.351} C_VEL
LIN {X 0,Y 406.221,Z 498.793,A -85,B 0,C 180,E1 -10875.381,E2 -10875.381} C_VEL
LIN {X 0,Y 405.245,Z 509.372,A -85,B 0,C 180,E1 -10876.557,E2 -10876.557} C_VEL
LIN {X 0,Y 404.586,Z 519.597,A -85,B 0,C 180,E1 -10877.968,E2 -10877.968} C_VEL
LIN {X 0,Y 403.83,Z 528.354,A -85,B 0,C 180,E1 -10879.47,E2 -10879.47} C_VEL
LIN {X 0,Y 403.407,Z 535.443,A -85,B 0,C 180,E1 -10880.978,E2 -10880.978} C_VEL
LIN {X 0,Y 403.124,Z 541.117,A -85,B 0,C 180,E1 -10882.486,E2 -10882.486} C_VEL
LIN {X 0,Y 402.939,Z 545.557,A -85,B 0,C 180,E1 -10883.992,E2 -10883.992} C_VEL
LIN {X 0,Y 402.939,Z 547.892,A -85,B 0,C 180,E1 -10884.996,E2 -10884.996} C_VEL
LIN {X 0,Y 402.863,Z 549.729,A -85,B 0,C 180,E1 -10885.998,E2 -10885.998} C_VEL
LIN {X 0,Y 402.868,Z 551.14,A -85,B 0,C 180,E1 -10886.999,E2 -10886.999} C_VEL
LIN {X 0,Y 402.946,Z 552.117,A -85,B 0,C 180,E1 -10888,E2 -10888} C_VEL
LIN {X 0,Y 402.904,Z 552.613,A -85,B 0,C 180,E1 -10889,E2 -10889} C_VEL
LIN {X 0,Y 402.906,Z 552.69,A -85,B 0,C 180,E1 -10889.999,E2 -10889.999} C_VEL
LIN {X 0,Y 402.904,Z 552.346,A -85,B 0,C 180,E1 -10890.998,E2 -10890.998} C_VEL
LIN {X 0,Y 402.952,Z 551.54,A -85,B 0,C 180,E1 -10891.998,E2 -10891.998} C_VEL
LIN {X 0,Y 402.926,Z 550.272,A -85,B 0,C 180,E1 -10892.998,E2 -10892.998} C_VEL
LIN {X 0,Y 402.939,Z 547.53,A -85,B 0,C 180,E1 -10894.501,E2 -10894.501} C_VEL
LIN {X 0,Y 402.99,Z 542.977,A -85,B 0,C 180,E1 -10896.247,E2 -10896.247} C_VEL
LIN {X 0,Y 403.192,Z 537.35,A -85,B 0,C 180,E1 -10898.015,E2 -10898.015} C_VEL
LIN {X 0,Y 403.463,Z 531.218,A -85,B 0,C 180,E1 -10899.524,E2 -10899.524} C_VEL
LIN {X 0,Y 403.912,Z 523.582,A -85,B 0,C 180,E1 -10901.033,E2 -10901.033} C_VEL
LIN {X 0,Y 404.597,Z 515.749,A -85,B 0,C 180,E1 -10902.285,E2 -10902.285} C_VEL
LIN {X 0,Y 405.317,Z 505.904,A -85,B 0,C 180,E1 -10903.567,E2 -10903.567} C_VEL
LIN {X 0,Y 406.019,Z 495.497,A -85,B 0,C 180,E1 -10904.663,E2 -10904.663} C_VEL
LIN {X 0,Y 406.713,Z 485.161,A -85,B 0,C 180,E1 -10905.535,E2 -10905.535} C_VEL
LIN {X 0,Y 407.524,Z 472.723,A -85,B 0,C 180,E1 -10906.338,E2 -10906.338} C_VEL
LIN {X 0,Y 408.193,Z 459.603,A -85,B 0,C 180,E1 -10906.954,E2 -10906.954} C_VEL
LIN {X 0,Y 408.674,Z 447.606,A -85,B 0,C 180,E1 -10907.32,E2 -10907.32} C_VEL
LIN {X 0,Y 409.499,Z 367.959,A -85,B 0,C 180,E1 -10908.734,E2 -10908.734} C_VEL
LIN {X 0,Y 405.541,Z 340.026,A -85,B 0,C 180,E1 -10909.453,E2 -10909.453} C_VEL
LIN {X 0,Y 406.595,Z 323.89,A -85,B 0,C 180,E1 -10912.617,E2 -10912.617} C_VEL
LIN {X 0,Y 407.46,Z 311.866,A -85,B 0,C 180,E1 -10914.997,E2 -10914.997} C_VEL
LIN {X 0,Y 405.424,Z 300.921,A -85,B 0,C 180,E1 -10917.331,E2 -10917.331} C_VEL
LIN {X 0,Y 404.24,Z 295.133,A -85,B 0,C 180,E1 -10918.631,E2 -10918.631} C_VEL
LIN {X 0,Y 404.138,Z 295.142,A -85,B 0,C 180,E1 -10922.62,E2 -10922.62} C_VEL
LIN {X 0,Y 404.177,Z 295.136,A -85,B 0,C 180,E1 -10925.189,E2 -10925.189} C_VEL
LIN {X 0,Y 404.144,Z 295.14,A -85,B 0,C 180,E1 -10928.757,E2 -10928.757} C_VEL
LIN {X 0,Y 404.114,Z 295.147,A -85,B 0,C 180,E1 -10931.598,E2 -10931.598} C_VEL
LIN {X 0,Y 404.139,Z 295.141,A -85,B 0,C 180,E1 -10934.521,E2 -10934.521} C_VEL
LIN {X 0,Y 404.125,Z 295.144,A -85,B 0,C 180,E1 -10937.294,E2 -10937.294} C_VEL
LIN {X 0,Y 404.126,Z 295.146,A -85,B 0,C 180,E1 -10939.95,E2 -10939.95} C_VEL
LIN {X 0,Y 404.128,Z 295.143,A -85,B 0,C 180,E1 -10943.125,E2 -10943.125} C_VEL
LIN {X 0,Y 404.137,Z 295.143,A -85,B 0,C 180,E1 -10946.187,E2 -10946.187} C_VEL
LIN {X 0,Y 404.136,Z 295.146,A -85,B 0,C 180,E1 -10949.714,E2 -10949.714} C_VEL
LIN {X 0,Y 404.098,Z 295.148,A -85,B 0,C 180,E1 -10953.116,E2 -10953.116} C_VEL
LIN {X 0,Y 404.145,Z 295.14,A -85,B 0,C 180,E1 -10956.424,E2 -10956.424} C_VEL
LIN {X 0,Y 404.183,Z 295.138,A -85,B 0,C 180,E1 -10959.874,E2 -10959.874} C_VEL
LIN {X 0,Y 404.207,Z 295.135,A -85,B 0,C 180,E1 -10962.993,E2 -10962.993} C_VEL
LIN {X 0,Y 404.274,Z 295.127,A -85,B 0,C 180,E1 -10966.939,E2 -10966.939} C_VEL
LIN {X 0,Y 404.245,Z 295.129,A -85,B 0,C 180,E1 -10969.988,E2 -10969.988} C_VEL
LIN {X 0,Y 404.327,Z 295.122,A -85,B 0,C 180,E1 -10973.011,E2 -10973.011} C_VEL
LIN {X 0,Y 404.246,Z 295.132,A -85,B 0,C 180,E1 -10975.013,E2 -10975.013} C_VEL
LIN {X 0,Y 404.464,Z 295.101,A -85,B 0,C 180,E1 -10978.008,E2 -10978.008} C_VEL
LIN {X 0,Y 404.459,Z 295.102,A -85,B 0,C 180,E1 -10981.992,E2 -10981.992} C_VEL
LIN {X 0,Y 404.326,Z 295.119,A -85,B 0,C 180,E1 -10986.604,E2 -10986.604} C_VEL
LIN {X 0,Y 404.255,Z 295.131,A -85,B 0,C 180,E1 -10989.002,E2 -10989.002} C_VEL
LIN {X 0,Y 404.246,Z 295.128,A -85,B 0,C 180,E1 -10992.042,E2 -10992.042} C_VEL
LIN {X 0,Y 404.196,Z 295.138,A -85,B 0,C 180,E1 -10995.118,E2 -10995.118} C_VEL
LIN {X 0,Y 404.195,Z 295.135,A -85,B 0,C 180,E1 -10998.239,E2 -10998.239} C_VEL
LIN {X 0,Y 404.13,Z 295.144,A -85,B 0,C 180,E1 -11001.42,E2 -11001.42} C_VEL
LIN {X 0,Y 404.156,Z 295.143,A -85,B 0,C 180,E1 -11004.667,E2 -11004.667} C_VEL
LIN {X 0,Y 404.159,Z 295.14,A -85,B 0,C 180,E1 -11008.003,E2 -11008.003} C_VEL
LIN {X 0,Y 404.132,Z 295.142,A -85,B 0,C 180,E1 -11011.559,E2 -11011.559} C_VEL
LIN {X 0,Y 404.178,Z 295.139,A -85,B 0,C 180,E1 -11015.017,E2 -11015.017} C_VEL
LIN {X 0,Y 404.142,Z 295.145,A -85,B 0,C 180,E1 -11018.759,E2 -11018.759} C_VEL
LIN {X 0,Y 404.113,Z 295.145,A -85,B 0,C 180,E1 -11021.6,E2 -11021.6} C_VEL
LIN {X 0,Y 404.14,Z 295.145,A -85,B 0,C 180,E1 -11024.523,E2 -11024.523} C_VEL
LIN {X 0,Y 404.131,Z 295.142,A -85,B 0,C 180,E1 -11027.297,E2 -11027.297} C_VEL
LIN {X 0,Y 404.165,Z 295.141,A -85,B 0,C 180,E1 -11029.956,E2 -11029.956} C_VEL
LIN {X 0,Y 404.132,Z 295.142,A -85,B 0,C 180,E1 -11033.126,E2 -11033.126} C_VEL
LIN {X 0,Y 404.141,Z 295.145,A -85,B 0,C 180,E1 -11036.189,E2 -11036.189} C_VEL
LIN {X 0,Y 404.143,Z 295.143,A -85,B 0,C 180,E1 -11039.716,E2 -11039.716} C_VEL
LIN {X 0,Y 404.193,Z 295.134,A -85,B 0,C 180,E1 -11043.124,E2 -11043.124} C_VEL
LIN {X 0,Y 404.176,Z 295.137,A -85,B 0,C 180,E1 -11045.336,E2 -11045.336} C_VEL
LIN {X 0,Y 404.163,Z 295.142,A -85,B 0,C 180,E1 -11048.583,E2 -11048.583} C_VEL
LIN {X 0,Y 404.235,Z 295.134,A -85,B 0,C 180,E1 -11050.025,E2 -11050.025} C_VEL
LIN {X 0,Y 405.031,Z 297.589,A -85,B 0,C 180,E1 -11050.2,E2 -11050.2} C_VEL
LIN {X 0,Y 408.124,Z 306.426,A -85,B 0,C 180,E1 -11050.521,E2 -11050.521} C_VEL
LIN {X 0,Y 410.598,Z 323.597,A -85,B 0,C 180,E1 -11050.958,E2 -11050.958} C_VEL
LIN {X 0,Y 409.434,Z 412.553,A -85,B 0,C 180,E1 -11052.552,E2 -11052.552} C_VEL
LIN {X 0,Y 409.101,Z 425.656,A -85,B 0,C 180,E1 -11052.989,E2 -11052.989} C_VEL
LIN {X 0,Y 408.445,Z 438.625,A -85,B 0,C 180,E1 -11053.636,E2 -11053.636} C_VEL
LIN {X 0,Y 407.824,Z 449.696,A -85,B 0,C 180,E1 -11054.381,E2 -11054.381} C_VEL
LIN {X 0,Y 407.162,Z 461.039,A -85,B 0,C 180,E1 -11055.366,E2 -11055.366} C_VEL
LIN {X 0,Y 406.366,Z 471.434,A -85,B 0,C 180,E1 -11056.499,E2 -11056.499} C_VEL
LIN {X 0,Y 405.582,Z 480.713,A -85,B 0,C 180,E1 -11057.746,E2 -11057.746} C_VEL
LIN {X 0,Y 404.853,Z 489.644,A -85,B 0,C 180,E1 -11059.246,E2 -11059.246} C_VEL
LIN {X 0,Y 404.205,Z 496.819,A -85,B 0,C 180,E1 -11060.746,E2 -11060.746} C_VEL
LIN {X 0,Y 403.704,Z 503.403,A -85,B 0,C 180,E1 -11062.499,E2 -11062.499} C_VEL
LIN {X 0,Y 403.427,Z 507.72,A -85,B 0,C 180,E1 -11064.001,E2 -11064.001} C_VEL
LIN {X 0,Y 403.151,Z 510.53,A -85,B 0,C 180,E1 -11065.29,E2 -11065.29} C_VEL
LIN {X 0,Y 403.134,Z 513.259,A -85,B 0,C 180,E1 -11067.003,E2 -11067.003} C_VEL
LIN {X 0,Y 402.91,Z 514.87,A -85,B 0,C 180,E1 -11069.002,E2 -11069.002} C_VEL
LIN {X 0,Y 402.889,Z 515.007,A -85,B 0,C 180,E1 -11069.583,E2 -11069.583} C_VEL
LIN {X 0,Y 402.238,Z 515.103,A -85,B 0,C 180,E1 -11070.418,E2 -11070.418} C_VEL
LIN {X 0,Y 399.444,Z 514.676,A -85,B 0,C 180,E1 -11071.775,E2 -11071.775} C_VEL
LIN {X 0,Y 397.095,Z 513.826,A -85,B 0,C 180,E1 -11072.866,E2 -11072.866} C_VEL
LIN {X 0,Y 396.11,Z 512.842,A -85,B 0,C 180,E1 -11073.702,E2 -11073.702} C_VEL
LIN {X 0,Y 396.043,Z 512.441,A -85,B 0,C 180,E1 -11073.984,E2 -11073.984} C_VEL
LIN {X 0,Y 396.24,Z 509.466,A -85,B 0,C 180,E1 -11075.599,E2 -11075.599} C_VEL
LIN {X 0,Y 396.515,Z 505.579,A -85,B 0,C 180,E1 -11077.128,E2 -11077.128} C_VEL
LIN {X 0,Y 396.897,Z 500.546,A -85,B 0,C 180,E1 -11078.658,E2 -11078.658} C_VEL
LIN {X 0,Y 397.519,Z 494.194,A -85,B 0,C 180,E1 -11080.184,E2 -11080.184} C_VEL
LIN {X 0,Y 398.199,Z 486.292,A -85,B 0,C 180,E1 -11081.712,E2 -11081.712} C_VEL
LIN {X 0,Y 398.951,Z 478.208,A -85,B 0,C 180,E1 -11082.981,E2 -11082.981} C_VEL
LIN {X 0,Y 399.871,Z 468.278,A -85,B 0,C 180,E1 -11084.245,E2 -11084.245} C_VEL
LIN {X 0,Y 400.592,Z 457.127,A -85,B 0,C 180,E1 -11085.389,E2 -11085.389} C_VEL
LIN {X 0,Y 401.321,Z 446.183,A -85,B 0,C 180,E1 -11086.273,E2 -11086.273} C_VEL
LIN {X 0,Y 401.959,Z 433.855,A -85,B 0,C 180,E1 -11087.03,E2 -11087.03} C_VEL
LIN {X 0,Y 402.538,Z 421.014,A -85,B 0,C 180,E1 -11087.595,E2 -11087.595} C_VEL
LIN {X 0,Y 402.811,Z 408.785,A -85,B 0,C 180,E1 -11087.943,E2 -11087.943} C_VEL
LIN {X 0,Y 403.787,Z 323.144,A -85,B 0,C 180,E1 -11089.488,E2 -11089.488} C_VEL
